FUNCTION "LAnyAxis_UnpubMoveJogPosAxis" : Void   // FC30008, SCL
TITLE = LAnyAxis_UnpubMoveJogPosAxis
{ S7_Optimized_Access := 'TRUE' }
AUTHOR : tech.team.motioncontrol@siemens.com
FAMILY : AnyAxis
VERSION : 1.0
// Support: tech.team.motioncontrol@siemens.com
   VAR_INPUT
      axis : TO_PositioningAxis;   // Axis specification
   END_VAR
   VAR_IN_OUT
      instMC : MC_MOVEJOG;   // Instance of MC_Instruction
   END_VAR
   // Ret_Val : No return value
BEGIN
   // Call of MC_Instruction
   #instMC(Axis := #axis);
END_FUNCTION

FUNCTION "LAnyAxis_UnpubMoveJogSyncAxis" : Void   // FC30010, SCL
TITLE = LAnyAxis_UnpubMoveJogSyncAxis
{ S7_Optimized_Access := 'TRUE' }
AUTHOR : tech.team.motioncontrol@siemens.com
FAMILY : AnyAxis
VERSION : 1.0
// Support: tech.team.motioncontrol@siemens.com
   VAR_INPUT
      axis : TO_SynchronousAxis;   // Axis specification
   END_VAR
   VAR_IN_OUT
      instMC : MC_MOVEJOG;   // Instance of MC_Instruction
   END_VAR
   // Ret_Val : No return value
BEGIN
   // Call of MC_Instruction
   #instMC(Axis := #axis);
END_FUNCTION

// folder: LAnyAxis_Blocks/InternalSubBlocks/MC_MoveRelative

FUNCTION "LAnyAxis_UnpubMoveRelativeSyncAxis" : Void   // FC30012, SCL
TITLE = LAnyAxis_UnpubMoveRelativeSyncAxis
{ S7_Optimized_Access := 'TRUE' }
AUTHOR : tech.team.motioncontrol@siemens.com
FAMILY : AnyAxis
VERSION : 1.0
// Support: tech.team.motioncontrol@siemens.com
   VAR_INPUT
      axis : TO_SynchronousAxis;   // Axis specification
   END_VAR
   VAR_IN_OUT
      instMC : MC_MOVERELATIVE;   // Instance of MC_Instruction
   END_VAR
   // Ret_Val : No return value
BEGIN
   // Call of MC_Instruction
   #instMC(Axis := #axis);
END_FUNCTION

// folder: LAnyAxis_Blocks/InternalSubBlocks/MC_MoveSuperimposed

FUNCTION "LAnyAxis_UnpubMoveSuperimposedSyncAxis" : Void   // FC30014, SCL
TITLE = LAnyAxis_UnpubMoveSuperimposedSyncAxis
{ S7_Optimized_Access := 'TRUE' }
AUTHOR : tech.team.motioncontrol@siemens.com
FAMILY : AnyAxis
VERSION : 1.0
// Support: tech.team.motioncontrol@siemens.com
   VAR_INPUT
      axis : TO_SynchronousAxis;   // Axis specification
   END_VAR
   VAR_IN_OUT
      instMC : MC_MOVESUPERIMPOSED;   // Instance of MC_Instruction
   END_VAR
   // Ret_Val : No return value
BEGIN
   // Call of MC_Instruction
   #instMC(Axis := #axis);
END_FUNCTION

// folder: LAnyAxis_Blocks/InternalSubBlocks/MC_MoveVelocity

FUNCTION "LAnyAxis_UnpubMoveVelocityPosAxis" : Void   // FC30015, SCL
TITLE = LAnyAxis_UnpubMoveVelocityPosAxis
{ S7_Optimized_Access := 'TRUE' }
AUTHOR : tech.team.motioncontrol@siemens.com
FAMILY : AnyAxis
VERSION : 1.0
// Support: tech.team.motioncontrol@siemens.com
   VAR_INPUT
      axis : TO_PositioningAxis;   // Axis specification
   END_VAR
   VAR_IN_OUT
      instMC : MC_MOVEVELOCITY;   // Instance of MC_Instruction
   END_VAR
   // Ret_Val : No return value
BEGIN
   // Call of MC_Instruction
   #instMC(Axis := #axis);
END_FUNCTION

FUNCTION "LAnyAxis_UnpubMoveVelocitySyncAxis" : Void   // FC30017, SCL
TITLE = LAnyAxis_UnpubMoveVelocitySyncAxis
{ S7_Optimized_Access := 'TRUE' }
AUTHOR : tech.team.motioncontrol@siemens.com
FAMILY : AnyAxis
VERSION : 1.0
// Support: tech.team.motioncontrol@siemens.com
   VAR_INPUT
      axis : TO_SynchronousAxis;   // Axis specification
   END_VAR
   VAR_IN_OUT
      instMC : MC_MOVEVELOCITY;   // Instance of MC_Instruction
   END_VAR
   // Ret_Val : No return value
BEGIN
   // Call of MC_Instruction
   #instMC(Axis := #axis);
END_FUNCTION

// folder: LAnyAxis_Blocks/InternalSubBlocks/MC_Power

FUNCTION "LAnyAxis_UnpubPowerExtEncoder" : Void   // FC30018, SCL
TITLE = LAnyAxis_UnpubPowerExtEncoder
{ S7_Optimized_Access := 'TRUE' }
AUTHOR : tech.team.motioncontrol@siemens.com
FAMILY : AnyAxis
VERSION : 1.0
// Support: tech.team.motioncontrol@siemens.com
   VAR_INPUT
      axis : TO_ExternalEncoder;   // Axis specification
   END_VAR
   VAR_IN_OUT
      instMC : MC_POWER;   // Instance of MC_Instruction
   END_VAR
   // Ret_Val : No return value
BEGIN
   // Call of MC_Instruction
   #instMC(Axis := #axis);
END_FUNCTION

FUNCTION "LAnyAxis_UnpubPowerPosAxis" : Void   // FC30019, SCL
TITLE = LAnyAxis_UnpubPowerPosAxis
{ S7_Optimized_Access := 'TRUE' }
AUTHOR : tech.team.motioncontrol@siemens.com
FAMILY : AnyAxis
VERSION : 1.0
// Support: tech.team.motioncontrol@siemens.com
   VAR_INPUT
      axis : TO_PositioningAxis;   // Axis specification
   END_VAR
   VAR_IN_OUT
      instMC : MC_POWER;   // Instance of MC_Instruction
   END_VAR
   // Ret_Val : No return value
BEGIN
   // Call of MC_Instruction
   #instMC(Axis := #axis);
END_FUNCTION

FUNCTION "LAnyAxis_UnpubPowerSpeedAxis" : Void   // FC30020, SCL
TITLE = LAnyAxis_UnpubPowerSpeedAxis
{ S7_Optimized_Access := 'TRUE' }
AUTHOR : tech.team.motioncontrol@siemens.com
FAMILY : AnyAxis
VERSION : 1.0
// Support: tech.team.motioncontrol@siemens.com
   VAR_INPUT
      axis : TO_SpeedAxis;   // Axis specification
   END_VAR
   VAR_IN_OUT
      instMC : MC_POWER;   // Instance of MC_Instruction
   END_VAR
   // Ret_Val : No return value
BEGIN
   // Call of MC_Instruction
   #instMC(Axis := #axis);
END_FUNCTION

FUNCTION "LAnyAxis_UnpubPowerSyncAxis" : Void   // FC30021, SCL
TITLE = LAnyAxis_UnpubPowerSyncAxis
{ S7_Optimized_Access := 'TRUE' }
AUTHOR : tech.team.motioncontrol@siemens.com
FAMILY : AnyAxis
VERSION : 1.0
// Support: tech.team.motioncontrol@siemens.com
   VAR_INPUT
      axis : TO_SynchronousAxis;   // Axis specification
   END_VAR
   VAR_IN_OUT
      instMC : MC_POWER;   // Instance of MC_Instruction
   END_VAR
   // Ret_Val : No return value
BEGIN
   // Call of MC_Instruction
   #instMC(Axis := #axis);
END_FUNCTION

// folder: LAnyAxis_Blocks/InternalSubBlocks/MC_Reset

FUNCTION "LAnyAxis_UnpubResetExtEncoder" : Void   // FC30022, SCL
TITLE = LAnyAxis_UnpubResetExtEncoder
{ S7_Optimized_Access := 'TRUE' }
AUTHOR : tech.team.motioncontrol@siemens.com
FAMILY : AnyAxis
VERSION : 1.0
// Support: tech.team.motioncontrol@siemens.com
   VAR_INPUT
      axis : TO_ExternalEncoder;   // Axis specification
   END_VAR
   VAR_IN_OUT
      instMC : MC_RESET;   // Instance of MC_Instruction
   END_VAR
   // Ret_Val : No return value
BEGIN
   // Call of MC_Instruction
   #instMC(Axis := #axis);
END_FUNCTION

FUNCTION "LAnyAxis_UnpubResetSpeedAxis" : Void   // FC30024, SCL
TITLE = LAnyAxis_UnpubResetSpeedAxis
{ S7_Optimized_Access := 'TRUE' }
AUTHOR : tech.team.motioncontrol@siemens.com
FAMILY : AnyAxis
VERSION : 1.0
// Support: tech.team.motioncontrol@siemens.com
   VAR_INPUT
      axis : TO_SpeedAxis;   // Axis specification
   END_VAR
   VAR_IN_OUT
      instMC : MC_RESET;   // Instance of MC_Instruction
   END_VAR
   // Ret_Val : No return value
BEGIN
   // Call of MC_Instruction
   #instMC(Axis := #axis);
END_FUNCTION

FUNCTION "LAnyAxis_UnpubResetSyncAxis" : Void   // FC30025, SCL
TITLE = LAnyAxis_UnpubResetSyncAxis
{ S7_Optimized_Access := 'TRUE' }
AUTHOR : tech.team.motioncontrol@siemens.com
FAMILY : AnyAxis
VERSION : 1.0
// Support: tech.team.motioncontrol@siemens.com
   VAR_INPUT
      axis : TO_SynchronousAxis;   // Axis specification
   END_VAR
   VAR_IN_OUT
      instMC : MC_RESET;   // Instance of MC_Instruction
   END_VAR
   // Ret_Val : No return value
BEGIN
   // Call of MC_Instruction
   #instMC(Axis := #axis);
END_FUNCTION

FUNCTION "LAnyAxis_UnpubResetProxy" : Void   // FC30057, SCL
TITLE = LAnyAxis_UnpubResetProxy
{ S7_Optimized_Access := 'TRUE' }
AUTHOR : tech.team.motioncontrol@siemens.com
FAMILY : AnyAxis
VERSION : 1.0
// Support: tech.team.motioncontrol@siemens.com
   VAR_INPUT
      axis : TO_LeadingAxisProxy;   // Axis specification
   END_VAR
   VAR_IN_OUT
      instMC : MC_RESET;   // Instance of MC_Instruction
   END_VAR
   // Ret_Val : No return value
BEGIN
   // Call of MC_Instruction
   #instMC(Axis := #axis);
END_FUNCTION

FUNCTION "LAnyAxis_UnpubResetPosAxis" : Void   // FC30071, SCL
TITLE = LAnyAxis_UnpubResetPosAxis
{ S7_Optimized_Access := 'TRUE' }
AUTHOR : tech.team.motioncontrol@siemens.com
FAMILY : AnyAxis
VERSION : 1.0
// Support: tech.team.motioncontrol@siemens.com
   VAR_INPUT
      axis : TO_PositioningAxis;   // Axis specification
   END_VAR
   VAR_IN_OUT
      instMC : MC_RESET;   // Instance of MC_Instruction
   END_VAR
   // Ret_Val : No return value
BEGIN
   // Call of MC_Instruction
   #instMC(Axis := #axis);
END_FUNCTION

// folder: LAnyAxis_Blocks/InternalSubBlocks/MC_SetAxisSTW

FUNCTION "LAnyAxis_UnpubSetAxisSTWPosAxis" : Void   // FC30026, SCL
TITLE = LAnyAxis_UnpubSetAxisSTWPosAxis
{ S7_Optimized_Access := 'TRUE' }
AUTHOR : tech.team.motioncontrol@siemens.com
FAMILY : AnyAxis
VERSION : 1.0
// Support: tech.team.motioncontrol@siemens.com
   VAR_INPUT
      axis : TO_PositioningAxis;   // Axis specification
   END_VAR
   VAR_IN_OUT
      instMC : MC_SETAXISSTW;   // Instance of MC_Instruction
   END_VAR
   // Ret_Val : No return value
BEGIN
   // Call of MC_Instruction
   #instMC(Axis := #axis);
END_FUNCTION

FUNCTION "LAnyAxis_UnpubSetAxisSTWSyncAxis" : Void   // FC30028, SCL
TITLE = LAnyAxis_UnpubSetAxisSTWSyncAxis
{ S7_Optimized_Access := 'TRUE' }
AUTHOR : tech.team.motioncontrol@siemens.com
FAMILY : AnyAxis
VERSION : 1.0
// Support: tech.team.motioncontrol@siemens.com
   VAR_INPUT
      axis : TO_SynchronousAxis;   // Axis specification
   END_VAR
   VAR_IN_OUT
      instMC : MC_SETAXISSTW;   // Instance of MC_Instruction
   END_VAR
   // Ret_Val : No return value
BEGIN
   // Call of MC_Instruction
   #instMC(Axis := #axis);
END_FUNCTION

// folder: LAnyAxis_Blocks/LAnyAxis_MC_SynchronousMotion

FUNCTION_BLOCK "LAnyAxis_MC_GearIn"   // FB30020, SCL
TITLE = LAnyAxis_MC_GearIn
{ S7_Optimized_Access := 'TRUE' }
AUTHOR : tech.team.motioncontrol@siemens.com
FAMILY : AnyAxis
VERSION : 1.0
// Support: tech.team.motioncontrol@siemens.com 
// See corresponding MC_ instruction in TIA Portal help (information system)
   VAR_INPUT
      Master : DB_ANY;   // See corresponding parameter of MC_ instruction in TIA Portal help (information system)
      Slave : DB_ANY;   // See corresponding parameter of MC_ instruction in TIA Portal help (information system)
      Execute : Bool;   // See corresponding parameter of MC_ instruction in TIA Portal help (information system)
      RatioNumerator : DInt := 1;   // See corresponding parameter of MC_ instruction in TIA Portal help (information system)
      RatioDenominator : DInt := 1;   // See corresponding parameter of MC_ instruction in TIA Portal help (information system)
      Acceleration : LReal := -1.0;   // See corresponding parameter of MC_ instruction in TIA Portal help (information system)
      Deceleration : LReal := -1.0;   // See corresponding parameter of MC_ instruction in TIA Portal help (information system)
      Jerk : LReal := -1.0;   // See corresponding parameter of MC_ instruction in TIA Portal help (information system)
   END_VAR
   VAR_OUTPUT
      InGear : Bool;   // See corresponding parameter of MC_ instruction in TIA Portal help (information system)
      Busy : Bool;   // See corresponding parameter of MC_ instruction in TIA Portal help (information system)
      CommandAborted : Bool;   // See corresponding parameter of MC_ instruction in TIA Portal help (information system)
      Error : Bool;   // See corresponding parameter of MC_ instruction in TIA Portal help (information system)
      ErrorID : Word;   // See corresponding parameter of MC_ instruction in TIA Portal help (information system)
   END_VAR
   VAR
      instMC : MC_GEARIN;   // Instance of MC_Instruction
      statExecuteOld : Bool;   // Old value of execute
      statAxis : DB_ANY;   // Internal variable of axis
      statAxisType : Int;   // Actual state / axis type
      statMaster : DB_ANY;   // Internal variable of Master
      statMasterType : Int;   // Type of master axis
   END_VAR
   VAR CONSTANT
      ERROR_INVALID_TECHNOLOGY_OBJECT : Word := 16#8002;   // See corresponding parameter of MC_ instruction in TIA Portal help (information system)
      IDLE : Int := 0;   // State idle
      INVALID_AXIS : Int := -1;   // Axis type: Invalid
      INVALID_MASTER : Int := -2;   // Invalid master type
      EXTERNAL_ENCODER : Int := 1;   // Axis type: External encoder
      POSITIONING_AXIS : Int := 3;   // Axis type: Positioning axis
      SYNCHRONOUS_AXIS : Int := 4;   // Axis type: Synchronous axis
      PROXY : Int := 5;   // Axis type: Leading axis proxy
   END_VAR
BEGIN
   REGION HEADER
     //================================================================================
     // SIEMENS AG
     // (c)Copyright 2020 All Rights Reserved
     //--------------------------------------------------------------------------------
     // Library: LAnyAxis 
     // Tested with: S7-1515T-2 PN
     // Engineering: TIA Portal V16
     // Restrictions: -
     // Requirements: S7-1500T FW 2.8.1
     // Functionality: Conversion DB_ANY --> TO_Axis
     // Support: tech.team.motioncontrol@siemens.com
     // Note: Parameter comments are only available in language 'English (United States)'
     //--------------------------------------------------------------------------------
     // Change log table:
     // Version  Date        Expert in charge  Changes applied
     // 01.00.00 10.03.2020  RS                First released version
     //================================================================================
   END_REGION

   REGION EXECUTE
     IF #Execute AND NOT #statExecuteOld THEN
       // Copy parameter
       #instMC.RatioNumerator := #RatioNumerator;
       #instMC.RatioDenominator := #RatioDenominator;
       #instMC.Acceleration := #Acceleration;
       #instMC.Deceleration := #Deceleration;
       #instMC.Jerk := #Jerk;

       // Check axis type
       CASE TypeOfDB(#Slave) OF
         TO_SYNCHRONOUSAXIS:
           #statAxisType := #SYNCHRONOUS_AXIS;
           #statAxis := #Slave;

           // Check master type
           CASE TypeOfDB(#Master) OF
             TO_POSITIONINGAXIS:
               #statMasterType := #POSITIONING_AXIS;
               #statMaster := #Master;

             TO_SYNCHRONOUSAXIS:
               #statMasterType := #SYNCHRONOUS_AXIS;
               #statMaster := #Master;

             TO_EXTERNALENCODER:
               #statMasterType := #EXTERNAL_ENCODER;
               #statMaster := #Master;

             TO_LEADINGAXISPROXY:
               #statMasterType := #PROXY;
               #statMaster := #Master;
             ELSE
               // Invalid master
               #statMasterType := #INVALID_AXIS;
               #statMaster := 0;

               #statAxisType := #INVALID_MASTER;
           END_CASE;

         ELSE
           #statAxisType := #INVALID_AXIS;
           #statAxis := 0;
       END_CASE;

     ELSIF NOT #Execute AND (#statAxisType < #IDLE) THEN
       #statAxisType := #IDLE;

       // Outputs
       #InGear := FALSE;
       #Busy := FALSE;
       #CommandAborted := FALSE;
       #Error := FALSE;
       #ErrorID := 16#0000;
     END_IF;

     // Edge detection
     #statExecuteOld := #Execute;
   END_REGION

   CASE #statAxisType OF
     #IDLE:
       ;

     #SYNCHRONOUS_AXIS:
       REGION VALID_AXIS
         // Inputs
         #instMC.Execute := #Execute;

         // Call of MC instruction
         CASE #statMasterType OF
           #POSITIONING_AXIS:
             "LAnyAxis_UnpubGearInMasterPosAxis"(slave := #statAxis,
                                                 master := #statMaster,
                                                 instMC := #instMC);
           #SYNCHRONOUS_AXIS:
             "LAnyAxis_UnpubGearInMasterSyncAxis"(slave := #statAxis,
                                                  master := #statMaster,
                                                  instMC := #instMC);
           #EXTERNAL_ENCODER:
             "LAnyAxis_UnpubGearInMasterExtEncoder"(slave := #statAxis,
                                                    master := #statMaster,
                                                    instMC := #instMC);
           #PROXY:
             "LAnyAxis_UnpubGearInMasterProxy"(slave := #statAxis,
                                               master := #statMaster,
                                               instMC := #instMC);
         END_CASE;

         // Outputs
         #InGear := #instMC.InGear;
         #Busy := #instMC.Busy;
         #CommandAborted := #instMC.CommandAborted;
         #Error := #instMC.Error;
         #ErrorID := #instMC.ErrorId;

         // Status of MC instruction
         IF NOT #instMC.Busy
           AND NOT #instMC.CommandAborted
           AND NOT #instMC.Error
         THEN
           // Not active
           #statAxisType := #IDLE;
         END_IF;
       END_REGION

     ELSE
       REGION INVALID_TECHNOLOGY_OBJECT
         // Outputs
         #InGear := FALSE;
         #Busy := FALSE;
         #CommandAborted := FALSE;
         #Error := TRUE;
         #ErrorID := #ERROR_INVALID_TECHNOLOGY_OBJECT;
       END_REGION
   END_CASE;
END_FUNCTION_BLOCK

FUNCTION_BLOCK "LAnyAxis_MC_GearInPos"   // FB30021, SCL
TITLE = LAnyAxis_MC_GearInPos
{ S7_Optimized_Access := 'TRUE' }
AUTHOR : tech.team.motioncontrol@siemens.com
FAMILY : AnyAxis
VERSION : 1.0
// Support: tech.team.motioncontrol@siemens.com 
// See corresponding MC_ instruction in TIA Portal help (information system)
   VAR_INPUT
      Master : DB_ANY;   // See corresponding parameter of MC_ instruction in TIA Portal help (information system)
      Slave : DB_ANY;   // See corresponding parameter of MC_ instruction in TIA Portal help (information system)
      Execute : Bool;   // See corresponding parameter of MC_ instruction in TIA Portal help (information system)
      RatioNumerator : DInt := 1;   // See corresponding parameter of MC_ instruction in TIA Portal help (information system)
      RatioDenominator : DInt := 1;   // See corresponding parameter of MC_ instruction in TIA Portal help (information system)
      MasterSyncPosition : LReal;   // See corresponding parameter of MC_ instruction in TIA Portal help (information system)
      SlaveSyncPosition : LReal;   // See corresponding parameter of MC_ instruction in TIA Portal help (information system)
      SyncProfileReference : DInt := 1;   // See corresponding parameter of MC_ instruction in TIA Portal help (information system)
      MasterStartDistance : LReal := 1.0;   // See corresponding parameter of MC_ instruction in TIA Portal help (information system)
      Velocity : LReal := -1.0;   // See corresponding parameter of MC_ instruction in TIA Portal help (information system)
      Acceleration : LReal := -1.0;   // See corresponding parameter of MC_ instruction in TIA Portal help (information system)
      Deceleration : LReal := -1.0;   // See corresponding parameter of MC_ instruction in TIA Portal help (information system)
      Jerk : LReal := -1.0;   // See corresponding parameter of MC_ instruction in TIA Portal help (information system)
      SyncDirection : DInt := 3;   // See corresponding parameter of MC_ instruction in TIA Portal help (information system)
   END_VAR
   VAR_OUTPUT
      StartSync : Bool;   // See corresponding parameter of MC_ instruction in TIA Portal help (information system)
      InSync : Bool;   // See corresponding parameter of MC_ instruction in TIA Portal help (information system)
      Busy : Bool;   // See corresponding parameter of MC_ instruction in TIA Portal help (information system)
      CommandAborted : Bool;   // See corresponding parameter of MC_ instruction in TIA Portal help (information system)
      Error : Bool;   // See corresponding parameter of MC_ instruction in TIA Portal help (information system)
      ErrorID : Word;   // See corresponding parameter of MC_ instruction in TIA Portal help (information system)
   END_VAR
   VAR
      instMC : MC_GEARINPOS;   // Instance of MC_Instruction
      statExecuteOld : Bool;   // Old value of execute
      statAxis : DB_ANY;   // Internal variable of axis
      statAxisType : Int;   // Actual state / axis type
      statMaster : DB_ANY;   // Internal variable of Master
      statMasterType : Int;   // Type of master axis
   END_VAR
   VAR CONSTANT
      ERROR_INVALID_TECHNOLOGY_OBJECT : Word := 16#8002;   // See corresponding parameter of MC_ instruction in TIA Portal help (information system)
      IDLE : Int := 0;   // State idle
      INVALID_AXIS : Int := -1;   // Axis type: Invalid
      INVALID_MASTER : Int := -2;   // Invalid master type
      EXTERNAL_ENCODER : Int := 1;   // Axis type: External encoder
      POSITIONING_AXIS : Int := 3;   // Axis type: Positioning axis
      SYNCHRONOUS_AXIS : Int := 4;   // Axis type: Synchronous axis
      PROXY : Int := 5;   // Axis type: Leading axis proxy
   END_VAR
BEGIN
   REGION HEADER
     //================================================================================
     // SIEMENS AG
     // (c)Copyright 2020 All Rights Reserved
     //--------------------------------------------------------------------------------
     // Library: LAnyAxis 
     // Tested with: S7-1515T-2 PN
     // Engineering: TIA Portal V16
     // Restrictions: -
     // Requirements: S7-1500T FW 2.8.1
     // Functionality: Conversion DB_ANY --> TO_Axis
     // Support: tech.team.motioncontrol@siemens.com
     // Note: Parameter comments are only available in language 'English (United States)'
     //--------------------------------------------------------------------------------
     // Change log table:
     // Version  Date        Expert in charge  Changes applied
     // 01.00.00 10.03.2020  RS                First released version
     //================================================================================
   END_REGION

   REGION EXECUTE
     IF #Execute AND NOT #statExecuteOld THEN
       // Copy parameter
       #instMC.RatioNumerator := #RatioNumerator;
       #instMC.RatioDenominator := #RatioDenominator;
       #instMC.MasterSyncPosition := #MasterSyncPosition;
       #instMC.SlaveSyncPosition := #SlaveSyncPosition;
       #instMC.SyncProfileReference := #SyncProfileReference;
       #instMC.MasterStartDistance := #MasterStartDistance;
       #instMC.Velocity := #Velocity;
       #instMC.Acceleration := #Acceleration;
       #instMC.Deceleration := #Deceleration;
       #instMC.Jerk := #Jerk;
       #instMC.SyncDirection := #SyncDirection;

       // Check axis type
       CASE TypeOfDB(#Slave) OF
         TO_SYNCHRONOUSAXIS:
           #statAxisType := #SYNCHRONOUS_AXIS;
           #statAxis := #Slave;

           // Check master type
           CASE TypeOfDB(#Master) OF
             TO_POSITIONINGAXIS:
               #statMasterType := #POSITIONING_AXIS;
               #statMaster := #Master;

             TO_SYNCHRONOUSAXIS:
               #statMasterType := #SYNCHRONOUS_AXIS;
               #statMaster := #Master;

             TO_EXTERNALENCODER:
               #statMasterType := #EXTERNAL_ENCODER;
               #statMaster := #Master;

             TO_LEADINGAXISPROXY:
               #statMasterType := #PROXY;
               #statMaster := #Master;
             ELSE
               #statMasterType := #INVALID_AXIS;
               #statMaster := 0;

               // Invalid master
               #statAxisType := #INVALID_MASTER;
           END_CASE;

         ELSE
           #statAxisType := #INVALID_AXIS;
           #statAxis := 0;
       END_CASE;

     ELSIF NOT #Execute AND (#statAxisType < #IDLE) THEN
       #statAxisType := #IDLE;

       // Outputs
       #StartSync := FALSE;
       #InSync := FALSE;
       #Busy := FALSE;
       #CommandAborted := FALSE;
       #Error := FALSE;
       #ErrorID := 16#0000;
     END_IF;

     // Edge detection
     #statExecuteOld := #Execute;
   END_REGION

   CASE #statAxisType OF
     #IDLE:
       ;

     #SYNCHRONOUS_AXIS:
       REGION VALID_AXIS
         // Inputs
         #instMC.Execute := #Execute;

         // Call of MC instruction
         CASE #statMasterType OF
           #POSITIONING_AXIS:
             "LAnyAxis_UnpubGearInPosMasterPosAxis"(slave := #statAxis,
                                                    master := #statMaster,
                                                    instMC := #instMC);
           #SYNCHRONOUS_AXIS:
             "LAnyAxis_UnpubGearInPosMasterSyncAxis"(slave := #statAxis,
                                                     master := #statMaster,
                                                     instMC := #instMC);
           #EXTERNAL_ENCODER:
             "LAnyAxis_UnpubGearInPosMasterExtEncoder"(slave := #statAxis,
                                                       master := #statMaster,
                                                       instMC := #instMC);
           #PROXY:
             "LAnyAxis_UnpubGearInPosMasterProxy"(slave := #statAxis,
                                                  master := #statMaster,
                                                  instMC := #instMC);
         END_CASE;

         // Outputs
         #StartSync := #instMC.StartSync;
         #InSync := #instMC.InSync;
         #Busy := #instMC.Busy;
         #CommandAborted := #instMC.CommandAborted;
         #Error := #instMC.Error;
         #ErrorID := #instMC.ErrorId;

         // Status of MC instruction
         IF NOT #instMC.Busy
           AND NOT #instMC.CommandAborted
           AND NOT #instMC.Error
         THEN
           // Not active
           #statAxisType := #IDLE;
         END_IF;
       END_REGION

     ELSE
       REGION INVALID_TECHNOLOGY_OBJECT
         // Outputs
         #StartSync := FALSE;
         #InSync := FALSE;
         #Busy := FALSE;
         #CommandAborted := FALSE;
         #Error := TRUE;
         #ErrorID := #ERROR_INVALID_TECHNOLOGY_OBJECT;
       END_REGION
   END_CASE;
END_FUNCTION_BLOCK

FUNCTION_BLOCK "LAnyAxis_MC_PhasingRelative"   // FB30022, SCL
TITLE = LAnyAxis_MC_PhasingRelative
{ S7_Optimized_Access := 'TRUE' }
AUTHOR : tech.team.motioncontrol@siemens.com
FAMILY : AnyAxis
VERSION : 1.1
// Support: tech.team.motioncontrol@siemens.com 
// See corresponding MC_ instruction in TIA Portal help (information system)
   VAR_INPUT
      Master : DB_ANY;   // See corresponding parameter of MC_ instruction in TIA Portal help (information system)
      Slave : DB_ANY;   // See corresponding parameter of MC_ instruction in TIA Portal help (information system)
      Execute : Bool;   // See corresponding parameter of MC_ instruction in TIA Portal help (information system)
      PhaseShift : LReal;   // See corresponding parameter of MC_ instruction in TIA Portal help (information system)
      Velocity : LReal := -1.0;   // See corresponding parameter of MC_ instruction in TIA Portal help (information system)
      Acceleration : LReal := -1.0;   // See corresponding parameter of MC_ instruction in TIA Portal help (information system)
      Deceleration : LReal := -1.0;   // See corresponding parameter of MC_ instruction in TIA Portal help (information system)
      Jerk : LReal := -1.0;   // See corresponding parameter of MC_ instruction in TIA Portal help (information system)
      ProfileReference : DInt;   // See corresponding parameter of MC_ instruction in TIA Portal help (information system)
      PhasingDistance : LReal;   // See corresponding parameter of MC_ instruction in TIA Portal help (information system)
      StartPosition : LReal;   // See corresponding parameter of MC_ instruction in TIA Portal help (information system)
      Direction : DInt := 3;   // See corresponding parameter of MC_ instruction in TIA Portal help (information system)
   END_VAR
   VAR_OUTPUT
      Done : Bool;   // See corresponding parameter of MC_ instruction in TIA Portal help (information system)
      Busy : Bool;   // See corresponding parameter of MC_ instruction in TIA Portal help (information system)
      CommandAborted : Bool;   // See corresponding parameter of MC_ instruction in TIA Portal help (information system)
      Error : Bool;   // See corresponding parameter of MC_ instruction in TIA Portal help (information system)
      ErrorID : Word;   // See corresponding parameter of MC_ instruction in TIA Portal help (information system)
      CoveredPhaseShift : LReal;   // See corresponding parameter of MC_ instruction in TIA Portal help (information system)
      StartPhasing : Bool;   // See corresponding parameter of MC_ instruction in TIA Portal help (information system)
   END_VAR
   VAR
      instMC : MC_PHASINGRELATIVE;   // Instance of MC_Instruction
      statExecuteOld : Bool;   // Old value of execute
      statAxis : DB_ANY;   // Internal variable of axis
      statAxisType : Int;   // Actual state / axis type
      statMaster : DB_ANY;   // Internal variable of Master
      statMasterType : Int;   // Type of master axis
   END_VAR
   VAR CONSTANT
      ERROR_INVALID_TECHNOLOGY_OBJECT : Word := 16#8002;   // See corresponding parameter of MC_ instruction in TIA Portal help (information system)
      IDLE : Int := 0;   // State idle
      INVALID_AXIS : Int := -1;   // Axis type: Invalid
      INVALID_MASTER : Int := -2;   // Invalid master type
      EXTERNAL_ENCODER : Int := 1;   // Axis type: External encoder
      POSITIONING_AXIS : Int := 3;   // Axis type: Positioning axis
      SYNCHRONOUS_AXIS : Int := 4;   // Axis type: Synchronous axis
      PROXY : Int := 5;   // Axis type: Leading axis proxy
   END_VAR
BEGIN
   REGION HEADER
     //================================================================================
     // SIEMENS AG
     // (c)Copyright 2021 All Rights Reserved
     //--------------------------------------------------------------------------------
     // Library: LAnyAxis 
     // Tested with: S7-1515T-2 PN
     // Engineering: TIA Portal V17
     // Restrictions: -
     // Requirements: S7-1500T FW 2.9
     // Functionality: Conversion DB_ANY --> TO_Axis
     // Support: tech.team.motioncontrol@siemens.com
     // Note: Parameter comments are only available in language 'English (United States)'
     //--------------------------------------------------------------------------------
     // Change log table:
     // Version  Date        Expert in charge  Changes applied
     // 01.00.00 10.03.2020  RS                First released version
     // 01.01.00 24.02.2021  RS                Update MC V6.0
     //================================================================================
   END_REGION

   REGION EXECUTE
     IF #Execute AND NOT #statExecuteOld THEN
       // Copy parameter
       #instMC.PhaseShift       := #PhaseShift;
       #instMC.Velocity         := #Velocity;
       #instMC.Acceleration     := #Acceleration;
       #instMC.Deceleration     := #Deceleration;
       #instMC.Jerk             := #Jerk;
       #instMC.ProfileReference := #ProfileReference;
       #instMC.PhasingDistance  := #PhasingDistance;
       #instMC.StartPosition    := #StartPosition;
       #instMC.Direction        := #Direction;

       // Check axis type
       CASE TypeOfDB(#Slave) OF
         TO_SYNCHRONOUSAXIS:
           #statAxisType := #SYNCHRONOUS_AXIS;
           #statAxis := #Slave;

           // Check master type
           CASE TypeOfDB(#Master) OF
             TO_POSITIONINGAXIS:
               #statMasterType := #POSITIONING_AXIS;
               #statMaster := #Master;

             TO_SYNCHRONOUSAXIS:
               #statMasterType := #SYNCHRONOUS_AXIS;
               #statMaster := #Master;

             TO_EXTERNALENCODER:
               #statMasterType := #EXTERNAL_ENCODER;
               #statMaster := #Master;

             TO_LEADINGAXISPROXY:
               #statMasterType := #PROXY;
               #statMaster := #Master;
             ELSE
               #statMasterType := #INVALID_AXIS;
               #statMaster := 0;

               // Invalid master
               #statAxisType := #INVALID_MASTER;
           END_CASE;

         ELSE
           #statAxisType := #INVALID_AXIS;
           #statAxis := 0;
       END_CASE;

     ELSIF NOT #Execute AND (#statAxisType < #IDLE) THEN
       #statAxisType := #IDLE;

       // Outputs
       #Done              := FALSE;
       #Busy              := FALSE;
       #CommandAborted    := FALSE;
       #Error             := FALSE;
       #ErrorID           := 16#0000;
       #CoveredPhaseShift := 0.0;
       #StartPhasing      := FALSE;
     END_IF;

     // Edge detection
     #statExecuteOld := #Execute;
   END_REGION

   CASE #statAxisType OF
     #IDLE:
       ;

     #SYNCHRONOUS_AXIS:
       REGION VALID_AXIS
         // Inputs  
         #instMC.Execute := #Execute;

         // Call of MC instruction
         CASE #statMasterType OF
           #POSITIONING_AXIS:
             "LAnyAxis_UnpubPhasingRelativeMasterPosAxis"(slave  := #statAxis,
                                                          master := #statMaster,
                                                          instMC := #instMC);
           #SYNCHRONOUS_AXIS:
             "LAnyAxis_UnpubPhasingRelativeMasterSyncAxis"(slave  := #statAxis,
                                                           master := #statMaster,
                                                           instMC := #instMC);
           #EXTERNAL_ENCODER:
             "LAnyAxis_UnpubPhasingRelativeMasterExtEncoder"(slave  := #statAxis,
                                                             master := #statMaster,
                                                             instMC := #instMC);
           #PROXY:
             "LAnyAxis_UnpubPhasingRelativeMasterProxy"(slave  := #statAxis,
                                                        master := #statMaster,
                                                        instMC := #instMC);
         END_CASE;

         // Outputs
         #Done              := #instMC.Done;
         #Busy              := #instMC.Busy;
         #CommandAborted    := #instMC.CommandAborted;
         #Error             := #instMC.Error;
         #ErrorID           := #instMC.ErrorId;
         #CoveredPhaseShift := #instMC.CoveredPhaseShift;
         #StartPhasing      := #instMC.StartPhasing;

         // Status of MC instruction
         IF NOT #instMC.Done
           AND NOT #instMC.Busy
           AND NOT #instMC.CommandAborted
           AND NOT #instMC.Error
         THEN
           // Not active
           #statAxisType := #IDLE;
         END_IF;
       END_REGION

     ELSE
       REGION INVALID_TECHNOLOGY_OBJECT
         // Outputs
         #Done              := FALSE;
         #Busy              := FALSE;
         #CommandAborted    := FALSE;
         #Error             := TRUE;
         #ErrorID           := #ERROR_INVALID_TECHNOLOGY_OBJECT;
         #CoveredPhaseShift := 0.0;
         #StartPhasing      := FALSE;
       END_REGION
   END_CASE;
END_FUNCTION_BLOCK

FUNCTION_BLOCK "LAnyAxis_MC_PhasingAbsolute"   // FB30023, SCL
TITLE = LAnyAxis_MC_PhasingAbsolute
{ S7_Optimized_Access := 'TRUE' }
AUTHOR : tech.team.motioncontrol@siemens.com
FAMILY : AnyAxis
VERSION : 1.1
// Support: tech.team.motioncontrol@siemens.com 
// See corresponding MC_ instruction in TIA Portal help (information system)
   VAR_INPUT
      Master : DB_ANY;   // See corresponding parameter of MC_ instruction in TIA Portal help (information system)
      Slave : DB_ANY;   // See corresponding parameter of MC_ instruction in TIA Portal help (information system)
      Execute : Bool;   // See corresponding parameter of MC_ instruction in TIA Portal help (information system)
      PhaseShift : LReal;   // See corresponding parameter of MC_ instruction in TIA Portal help (information system)
      Velocity : LReal := -1.0;   // See corresponding parameter of MC_ instruction in TIA Portal help (information system)
      Acceleration : LReal := -1.0;   // See corresponding parameter of MC_ instruction in TIA Portal help (information system)
      Deceleration : LReal := -1.0;   // See corresponding parameter of MC_ instruction in TIA Portal help (information system)
      Jerk : LReal := -1.0;   // See corresponding parameter of MC_ instruction in TIA Portal help (information system)
      ProfileReference : DInt;   // See corresponding parameter of MC_ instruction in TIA Portal help (information system)
      PhasingDistance : LReal;   // See corresponding parameter of MC_ instruction in TIA Portal help (information system)
      StartPosition : LReal;   // See corresponding parameter of MC_ instruction in TIA Portal help (information system)
      Direction : DInt := 3;   // See corresponding parameter of MC_ instruction in TIA Portal help (information system)
   END_VAR
   VAR_OUTPUT
      Done : Bool;   // See corresponding parameter of MC_ instruction in TIA Portal help (information system)
      Busy : Bool;   // See corresponding parameter of MC_ instruction in TIA Portal help (information system)
      CommandAborted : Bool;   // See corresponding parameter of MC_ instruction in TIA Portal help (information system)
      Error : Bool;   // See corresponding parameter of MC_ instruction in TIA Portal help (information system)
      ErrorID : Word;   // See corresponding parameter of MC_ instruction in TIA Portal help (information system)
      AbsolutePhaseShift : LReal;   // See corresponding parameter of MC_ instruction in TIA Portal help (information system)
      StartPhasing : Bool;   // See corresponding parameter of MC_ instruction in TIA Portal help (information system)
   END_VAR
   VAR
      instMC : MC_PHASINGABSOLUTE;   // Instance of MC_Instruction
      statExecuteOld : Bool;   // Old value of execute
      statAxis : DB_ANY;   // Internal variable of axis
      statAxisType : Int;   // Actual state / axis type
      statMaster : DB_ANY;   // Internal variable of Master
      statMasterType : Int;   // Type of master axis
   END_VAR
   VAR CONSTANT
      ERROR_INVALID_TECHNOLOGY_OBJECT : Word := 16#8002;   // See corresponding parameter of MC_ instruction in TIA Portal help (information system)
      IDLE : Int := 0;   // State idle
      INVALID_AXIS : Int := -1;   // Axis type: Invalid
      INVALID_MASTER : Int := -2;   // Invalid master type
      EXTERNAL_ENCODER : Int := 1;   // Axis type: External encoder
      POSITIONING_AXIS : Int := 3;   // Axis type: Positioning axis
      SYNCHRONOUS_AXIS : Int := 4;   // Axis type: Synchronous axis
      PROXY : Int := 5;   // Axis type: Leading axis proxy
   END_VAR
BEGIN
   REGION HEADER
     //================================================================================
     // SIEMENS AG
     // (c)Copyright 2021 All Rights Reserved
     //--------------------------------------------------------------------------------
     // Library: LAnyAxis 
     // Tested with: S7-1515T-2 PN
     // Engineering: TIA Portal V17
     // Restrictions: -
     // Requirements: S7-1500T FW 2.9 
     // Functionality: Conversion DB_ANY --> TO_Axis
     // Support: tech.team.motioncontrol@siemens.com
     // Note: Parameter comments are only available in language 'English (United States)'
     //--------------------------------------------------------------------------------
     // Change log table:
     // Version  Date        Expert in charge  Changes applied
     // 01.00.00 10.03.2020  RS                First released version
     // 01.01.00 24.02.2021  RS                Update MC V6.0
     //================================================================================
   END_REGION

   REGION EXECUTE
     IF #Execute AND NOT #statExecuteOld THEN
       // Copy parameter
       #instMC.PhaseShift       := #PhaseShift;
       #instMC.Velocity         := #Velocity;
       #instMC.Acceleration     := #Acceleration;
       #instMC.Deceleration     := #Deceleration;
       #instMC.Jerk             := #Jerk;
       #instMC.ProfileReference := #ProfileReference;
       #instMC.PhasingDistance  := #PhasingDistance;
       #instMC.StartPosition    := #StartPosition;
       #instMC.Direction        := #Direction;

       // Check axis type
       CASE TypeOfDB(#Slave) OF
         TO_SYNCHRONOUSAXIS:
           #statAxisType := #SYNCHRONOUS_AXIS;
           #statAxis := #Slave;

           // Check master type
           CASE TypeOfDB(#Master) OF
             TO_POSITIONINGAXIS:
               #statMasterType := #POSITIONING_AXIS;
               #statMaster := #Master;

             TO_SYNCHRONOUSAXIS:
               #statMasterType := #SYNCHRONOUS_AXIS;
               #statMaster := #Master;

             TO_EXTERNALENCODER:
               #statMasterType := #EXTERNAL_ENCODER;
               #statMaster := #Master;

             TO_LEADINGAXISPROXY:
               #statMasterType := #PROXY;
               #statMaster := #Master;
             ELSE
               #statMasterType := #INVALID_AXIS;
               #statMaster := 0;

               // Invalid master
               #statAxisType := #INVALID_MASTER;
           END_CASE;

         ELSE
           #statAxisType := #INVALID_AXIS;
           #statAxis := 0;
       END_CASE;

     ELSIF NOT #Execute AND (#statAxisType < #IDLE) THEN
       #statAxisType := #IDLE;

       // Outputs
       #Done               := FALSE;
       #Busy               := FALSE;
       #CommandAborted     := FALSE;
       #Error              := FALSE;
       #ErrorID            := 16#0000;
       #AbsolutePhaseShift := 0.0;
       #StartPhasing       := FALSE;
     END_IF;

     // Edge detection
     #statExecuteOld := #Execute;
   END_REGION

   CASE #statAxisType OF
     #IDLE:
       ;

     #SYNCHRONOUS_AXIS:
       REGION VALID_AXIS
         // Inputs 
         #instMC.Execute := #Execute;

         // Call of MC instruction
         CASE #statMasterType OF
           #POSITIONING_AXIS:
             "LAnyAxis_UnpubPhasingAbsoluteMasterPosAxis"(slave := #statAxis,
                                                          master := #statMaster,
                                                          instMC := #instMC);
           #SYNCHRONOUS_AXIS:
             "LAnyAxis_UnpubPhasingAbsoluteMasterSyncAxis"(slave := #statAxis,
                                                           master := #statMaster,
                                                           instMC := #instMC);
           #EXTERNAL_ENCODER:
             "LAnyAxis_UnpubPhasingAbsoluteMasterExtEncoder"(slave := #statAxis,
                                                             master := #statMaster,
                                                             instMC := #instMC);
           #PROXY:
             "LAnyAxis_UnpubPhasingAbsoluteMasterProxy"(slave := #statAxis,
                                                        master := #statMaster,
                                                        instMC := #instMC);
         END_CASE;

         // Outputs
         #Done               := #instMC.Done;
         #Busy               := #instMC.Busy;
         #CommandAborted     := #instMC.CommandAborted;
         #Error              := #instMC.Error;
         #ErrorID            := #instMC.ErrorId;
         #AbsolutePhaseShift := #instMC.AbsolutePhaseShift;
         #StartPhasing       := #instMC.StartPhasing;

         // Status of MC instruction
         IF NOT #instMC.Done
           AND NOT #instMC.Busy
           AND NOT #instMC.CommandAborted
           AND NOT #instMC.Error
         THEN
           // Not active
           #statAxisType := #IDLE;
         END_IF;
       END_REGION

     ELSE
       REGION INVALID_TECHNOLOGY_OBJECT
         // Outputs
         #Done               := FALSE;
         #Busy               := FALSE;
         #CommandAborted     := FALSE;
         #Error              := TRUE;
         #ErrorID            := #ERROR_INVALID_TECHNOLOGY_OBJECT;
         #AbsolutePhaseShift := 0.0;
         #StartPhasing       := FALSE;
       END_REGION
   END_CASE;
END_FUNCTION_BLOCK

FUNCTION_BLOCK "LAnyAxis_MC_CamIn"   // FB30024, SCL
TITLE = LAnyAxis_MC_CamIn
{ S7_Optimized_Access := 'TRUE' }
AUTHOR : tech.team.motioncontrol@siemens.com
FAMILY : AnyAxis
VERSION : 1.1
// Support: tech.team.motioncontrol@siemens.com 
// See corresponding MC_ instruction in TIA Portal help (information system)
   VAR_INPUT
      Master : DB_ANY;   // See corresponding parameter of MC_ instruction in TIA Portal help (information system)
      Slave : DB_ANY;   // See corresponding parameter of MC_ instruction in TIA Portal help (information system)
      Cam : DB_ANY;   // See corresponding parameter of MC_ instruction in TIA Portal help (information system)
      Execute : Bool;   // See corresponding parameter of MC_ instruction in TIA Portal help (information system)
      MasterOffset : LReal;   // See corresponding parameter of MC_ instruction in TIA Portal help (information system)
      SlaveOffset : LReal;   // See corresponding parameter of MC_ instruction in TIA Portal help (information system)
      MasterScaling : LReal := 1.0;   // See corresponding parameter of MC_ instruction in TIA Portal help (information system)
      SlaveScaling : LReal := 1.0;   // See corresponding parameter of MC_ instruction in TIA Portal help (information system)
      MasterSyncPosition : LReal;   // See corresponding parameter of MC_ instruction in TIA Portal help (information system)
      SyncProfileReference : DInt := 1;   // See corresponding parameter of MC_ instruction in TIA Portal help (information system)
      MasterStartDistance : LReal;   // See corresponding parameter of MC_ instruction in TIA Portal help (information system)
      Velocity : LReal := -1.0;   // See corresponding parameter of MC_ instruction in TIA Portal help (information system)
      Acceleration : LReal := -1.0;   // See corresponding parameter of MC_ instruction in TIA Portal help (information system)
      Deceleration : LReal := -1.0;   // See corresponding parameter of MC_ instruction in TIA Portal help (information system)
      Jerk : LReal := -1.0;   // See corresponding parameter of MC_ instruction in TIA Portal help (information system)
      ApplicationMode : DInt;   // See corresponding parameter of MC_ instruction in TIA Portal help (information system)
      SyncDirection : DInt := 3;   // See corresponding parameter of MC_ instruction in TIA Portal help (information system)
   END_VAR
   VAR_OUTPUT
      StartSync : Bool;   // See corresponding parameter of MC_ instruction in TIA Portal help (information system)
      InSync : Bool;   // See corresponding parameter of MC_ instruction in TIA Portal help (information system)
      Busy : Bool;   // See corresponding parameter of MC_ instruction in TIA Portal help (information system)
      CommandAborted : Bool;   // See corresponding parameter of MC_ instruction in TIA Portal help (information system)
      Error : Bool;   // See corresponding parameter of MC_ instruction in TIA Portal help (information system)
      ErrorID : Word;   // See corresponding parameter of MC_ instruction in TIA Portal help (information system)
      EndOfProfile : Bool;   // See corresponding parameter of MC_ instruction in TIA Portal help (information system)
   END_VAR
   VAR
      instMC : MC_CAMIN;   // Instance of MC_Instruction
      statExecuteOld : Bool;   // Old value of execute
      statAxis : DB_ANY;   // Internal variable of axis
      statAxisType : Int;   // Actual state / axis type
      statMaster : DB_ANY;   // Internal variable of master
      statMasterType : Int;   // Type of master axis
      statCam : DB_ANY;   // Internal variable of cam
      statCamType : Int;   // Type of cam
   END_VAR
   VAR CONSTANT
      ERROR_INVALID_TECHNOLOGY_OBJECT : Word := 16#8002;   // See corresponding parameter of MC_ instruction in TIA Portal help (information system)
      IDLE : Int := 0;   // State idle
      INVALID_AXIS : Int := -1;   // Axis type: Invalid
      INVALID_MASTER : Int := -2;   // Invalid master type
      INVALID_CAM : Int := -3;   // Invalid cam
      EXTERNAL_ENCODER : Int := 1;   // Axis type: External encoder
      POSITIONING_AXIS : Int := 3;   // Axis type: Positioning axis
      SYNCHRONOUS_AXIS : Int := 4;   // Axis type: Synchronous axis
      CAM_1K : Int;   // Cam type: Cam
      CAM_10K : Int := 1;   // Cam type: Cam_10k
      PROXY : Int := 5;   // Axis type: Leading axis proxy
   END_VAR
BEGIN
   REGION HEADER
     //================================================================================
     // SIEMENS AG
     // (c)Copyright 2021 All Rights Reserved
     //--------------------------------------------------------------------------------
     // Library: LAnyAxis 
     // Tested with: S7-1515T-2 PN
     // Engineering: TIA Portal V17
     // Restrictions: -
     // Requirements: S7-1500T FW 2.9
     // Functionality: Conversion DB_ANY --> TO_Axis
     // Support: tech.team.motioncontrol@siemens.com
     // Note: Parameter comments are only available in language 'English (United States)'
     //--------------------------------------------------------------------------------
     // Change log table:
     // Version  Date        Expert in charge  Changes applied
     // 01.00.00 10.03.2020  RS                First released version
     // 01.01.00 24.02.2021  RS                Update MC V6.0
     //================================================================================
   END_REGION

   REGION EXECUTE
     IF #Execute AND NOT #statExecuteOld THEN
       // Copy parameter
       #instMC.MasterOffset         := #MasterOffset;
       #instMC.SlaveOffset          := #SlaveOffset;
       #instMC.MasterScaling        := #MasterScaling;
       #instMC.SlaveScaling         := #SlaveScaling;
       #instMC.MasterSyncPosition   := #MasterSyncPosition;
       #instMC.SyncProfileReference := #SyncProfileReference;
       #instMC.MasterStartDistance  := #MasterStartDistance;
       #instMC.Velocity             := #Velocity;
       #instMC.Acceleration         := #Acceleration;
       #instMC.Deceleration         := #Deceleration;
       #instMC.Jerk                 := #Jerk;
       #instMC.ApplicationMode      := #ApplicationMode;
       #instMC.SyncDirection        := #SyncDirection;

       // Check axis type
       CASE TypeOfDB(#Slave) OF
         TO_SYNCHRONOUSAXIS:
           #statAxisType := #SYNCHRONOUS_AXIS;
           #statAxis := #Slave;

           // Check master type
           CASE TypeOfDB(#Master) OF
             TO_POSITIONINGAXIS:
               #statMasterType := #POSITIONING_AXIS;
               #statMaster := #Master;

             TO_SYNCHRONOUSAXIS:
               #statMasterType := #SYNCHRONOUS_AXIS;
               #statMaster := #Master;

             TO_EXTERNALENCODER:
               #statMasterType := #EXTERNAL_ENCODER;
               #statMaster := #Master;

             TO_LEADINGAXISPROXY:
               #statMasterType := #PROXY;
               #statMaster := #Master;
             ELSE
               #statMasterType := #INVALID_AXIS;
               #statMaster := 0;

               // Invalid master
               #statAxisType := #INVALID_MASTER;
           END_CASE;

         ELSE
           #statAxisType := #INVALID_AXIS;
           #statAxis := 0;
       END_CASE;

       CASE TypeOfDB(#Cam) OF
         TO_CAM:
           #statCam := #Cam;
           #statCamType := #CAM_1K;

         TO_CAM_10K:
           #statCam := #Cam;
           #statCamType := #CAM_10K;

         ELSE
           #statCam := 0;
           #statAxisType := #INVALID_CAM;
       END_CASE;

     ELSIF NOT #Execute AND (#statAxisType < #IDLE) THEN
       #statAxisType := #IDLE;

       // Outputs
       #StartSync      := FALSE;
       #InSync         := FALSE;
       #Busy           := FALSE;
       #CommandAborted := FALSE;
       #Error          := FALSE;
       #ErrorID        := 16#0000;
       #EndOfProfile   := FALSE;
     END_IF;

     // Edge detection
     #statExecuteOld := #Execute;
   END_REGION

   CASE #statAxisType OF
     #IDLE:
       ;

     #SYNCHRONOUS_AXIS:
       REGION VALID_AXIS
         // Inputs 
         #instMC.Execute := #Execute;

         // Call of MC instruction
         CASE #statMasterType OF
           #POSITIONING_AXIS:
             CASE #statCamType OF
               #CAM_1K:
                 "LAnyAxis_UnpubCamInMasterPosAxis"(slave  := #statAxis,
                                                    master := #statMaster,
                                                    cam    := #statCam,
                                                    instMC := #instMC);
               #CAM_10K:
                 "LAnyAxis_UnpubCamIn10kMasterPosAxis"(slave  := #statAxis,
                                                       master := #statMaster,
                                                       cam    := #statCam,
                                                       instMC := #instMC);
             END_CASE;

           #SYNCHRONOUS_AXIS:
             CASE #statCamType OF
               #CAM_1K:
                 "LAnyAxis_UnpubCamInMasterSyncAxis"(slave  := #statAxis,
                                                     master := #statMaster,
                                                     cam    := #statCam,
                                                     instMC := #instMC);

               #CAM_10K:
                 "LAnyAxis_UnpubCamIn10kMasterSyncAxis"(slave  := #statAxis,
                                                        master := #statMaster,
                                                        cam    := #statCam,
                                                        instMC := #instMC);
             END_CASE;

           #EXTERNAL_ENCODER:
             CASE #statCamType OF
               #CAM_1K:
                 "LAnyAxis_UnpubCamInMasterExtEncoder"(slave  := #statAxis,
                                                       master := #statMaster,
                                                       cam    := #statCam,
                                                       instMC := #instMC);

               #CAM_10K:
                 "LAnyAxis_UnpubCamIn10kMasterExtEncoder"(slave  := #statAxis,
                                                          master := #statMaster,
                                                          cam    := #statCam,
                                                          instMC := #instMC);
             END_CASE;

           #PROXY:
             CASE #statCamType OF
               #CAM_1K:
                 "LAnyAxis_UnpubCamInMasterProxy"(slave  := #statAxis,
                                                  master := #statMaster,
                                                  cam    := #statCam,
                                                  instMC := #instMC);

               #CAM_10K:
                 "LAnyAxis_UnpubCamIn10kMasterProxy"(slave  := #statAxis,
                                                     master := #statMaster,
                                                     cam    := #statCam,
                                                     instMC := #instMC);
             END_CASE;
         END_CASE;

         // Outputs
         #StartSync      := #instMC.StartSync;
         #InSync         := #instMC.InSync;
         #Busy           := #instMC.Busy;
         #CommandAborted := #instMC.CommandAborted;
         #Error          := #instMC.Error;
         #ErrorID        := #instMC.ErrorId;
         #EndOfProfile   := #instMC.EndOfProfile;

         // Status of MC instruction
         IF NOT #instMC.Busy
           AND NOT #instMC.CommandAborted
           AND NOT #instMC.Error
           AND NOT #instMC.EndOfProfile
         THEN
           // Not active
           #statAxisType := #IDLE;
         END_IF;
       END_REGION
     ELSE
       REGION INVALID_TECHNOLOGY_OBJECT
         // Outputs
         #StartSync      := FALSE;
         #InSync         := FALSE;
         #Busy           := FALSE;
         #CommandAborted := FALSE;
         #Error          := TRUE;
         #ErrorID        := #ERROR_INVALID_TECHNOLOGY_OBJECT;
         #EndOfProfile   := FALSE;
       END_REGION
   END_CASE;
END_FUNCTION_BLOCK

FUNCTION_BLOCK "LAnyAxis_MC_SynchronizedMotionSimulation"   // FB30025, SCL
TITLE = LAnyAxis_MC_SynchronizedMotionSimulation
{ S7_Optimized_Access := 'TRUE' }
AUTHOR : tech.team.motioncontrol@siemens.com
FAMILY : AnyAxis
VERSION : 1.0
// Support: tech.team.motioncontrol@siemens.com 
// See corresponding MC_ instruction in TIA Portal help (information system)
   VAR_INPUT
      Slave : DB_ANY;   // See corresponding parameter of MC_ instruction in TIA Portal help (information system)
      Enable : Bool;   // See corresponding parameter of MC_ instruction in TIA Portal help (information system)
   END_VAR
   VAR_OUTPUT
      InSimulation : Bool;   // See corresponding parameter of MC_ instruction in TIA Portal help (information system)
      Busy : Bool;   // See corresponding parameter of MC_ instruction in TIA Portal help (information system)
      Error : Bool;   // See corresponding parameter of MC_ instruction in TIA Portal help (information system)
      ErrorID : Word;   // See corresponding parameter of MC_ instruction in TIA Portal help (information system)
   END_VAR
   VAR
      instMC : MC_SYNCHRONIZEDMOTIONSIMULATION;   // Instance of MC_Instruction
      statAxis : DB_ANY;   // Internal variable of axis
      statAxisType : Int;   // Actual state / axis type
   END_VAR
   VAR CONSTANT
      ERROR_INVALID_TECHNOLOGY_OBJECT : Word := 16#8002;   // See corresponding parameter of MC_ instruction in TIA Portal help (information system)
      IDLE : Int := 0;   // State idle
      INVALID_AXIS : Int := -1;   // Axis type: Invalid
      SYNCHRONOUS_AXIS : Int := 4;   // Axis type: Synchronous axis
   END_VAR
BEGIN
   REGION HEADER
     //================================================================================
     // SIEMENS AG
     // (c)Copyright 2020 All Rights Reserved
     //--------------------------------------------------------------------------------
     // Library: LAnyAxis 
     // Tested with: S7-1515T-2 PN
     // Engineering: TIA Portal V16
     // Restrictions: -
     // Requirements: S7-1500T FW 2.8.1
     // Functionality: Conversion DB_ANY --> TO_Axis
     // Support: tech.team.motioncontrol@siemens.com
     // Note: Parameter comments are only available in language 'English (United States)'
     //--------------------------------------------------------------------------------
     // Change log table:
     // Version  Date        Expert in charge  Changes applied
     // 01.00.00 10.03.2020  RS                First released version
     //================================================================================
   END_REGION

   REGION ENABLE
     IF (#statAxisType = #IDLE) AND #Enable THEN
       // check axis type
       CASE TypeOfDB(#Slave) OF
         TO_SYNCHRONOUSAXIS:
           #statAxisType := #SYNCHRONOUS_AXIS;
           #statAxis := #Slave;
         ELSE
           #statAxisType := #INVALID_AXIS;
           #statAxis := 0;
       END_CASE;

     ELSIF NOT #Enable AND (#statAxisType = #INVALID_AXIS) THEN
       #statAxisType := #IDLE;

       // Outputs
       #InSimulation := FALSE;
       #Busy := FALSE;
       #Error := FALSE;
       #ErrorID := 16#0000;
     END_IF;
   END_REGION

   CASE #statAxisType OF
     #IDLE:
       ;

     #SYNCHRONOUS_AXIS:
       REGION SYNCHRONOUS_AXIS
         // Inputs
         #instMC.Enable := #Enable;

         // Call of MC instruction
         #instMC(Slave := #statAxis);

         // Outputs
         #InSimulation := #instMC.InSimulation;
         #Busy := #instMC.Busy;
         #Error := #instMC.Error;
         #ErrorID := #instMC.ErrorId;

         // Status of MC instruction
         IF NOT #instMC.Busy
           AND NOT #instMC.Error
         THEN
           // Not active
           #statAxisType := #IDLE;
         END_IF;
       END_REGION

     ELSE
       REGION INVALID_AXIS
         // Outputs
         #InSimulation := FALSE;
         #Busy := FALSE;
         #Error := TRUE;
         #ErrorID := #ERROR_INVALID_TECHNOLOGY_OBJECT;
       END_REGION
   END_CASE;
END_FUNCTION_BLOCK

FUNCTION_BLOCK "LAnyAxis_MC_OffsetRelative"   // FB30028, SCL
TITLE = LAnyAxis_MC_OffsetRelative
{ S7_Optimized_Access := 'TRUE' }
AUTHOR : tech.team.motioncontrol@siemens.com
FAMILY : AnyAxis
VERSION : 1.1
// Support: tech.team.motioncontrol@siemens.com 
// See corresponding MC_ instruction in TIA Portal help (information system)
   VAR_INPUT
      Slave : DB_ANY;   // See corresponding parameter of MC_ instruction in TIA Portal help (information system)
      Execute : Bool;   // See corresponding parameter of MC_ instruction in TIA Portal help (information system)
      Offset : LReal;   // See corresponding parameter of MC_ instruction in TIA Portal help (information system)
      ProfileReference : DInt := 1;   // See corresponding parameter of MC_ instruction in TIA Portal help (information system)
      OffsetDistance : LReal;   // See corresponding parameter of MC_ instruction in TIA Portal help (information system)
      StartPosition : LReal;   // See corresponding parameter of MC_ instruction in TIA Portal help (information system)
      Direction : DInt := 3;   // See corresponding parameter of MC_ instruction in TIA Portal help (information system)
   END_VAR
   VAR_OUTPUT
      Done : Bool;   // See corresponding parameter of MC_ instruction in TIA Portal help (information system)
      Busy : Bool;   // See corresponding parameter of MC_ instruction in TIA Portal help (information system)
      CommandAborted : Bool;   // See corresponding parameter of MC_ instruction in TIA Portal help (information system)
      Error : Bool;   // See corresponding parameter of MC_ instruction in TIA Portal help (information system)
      ErrorID : Word;   // See corresponding parameter of MC_ instruction in TIA Portal help (information system)
      CoveredOffset : LReal;   // See corresponding parameter of MC_ instruction in TIA Portal help (information system)
      StartOffset : Bool;   // See corresponding parameter of MC_ instruction in TIA Portal help (information system)
   END_VAR
   VAR
      instMC : MC_OFFSETRELATIVE;   // Instance of MC_Instruction
      statExecuteOld : Bool;   // Old value of execute
      statAxis : DB_ANY;   // Internal variable of axis
      statAxisType : Int;   // Actual state / axis type
   END_VAR
   VAR CONSTANT
      ERROR_INVALID_TECHNOLOGY_OBJECT : Word := 16#8002;   // See corresponding parameter of MC_ instruction in TIA Portal help (information system)
      IDLE : Int := 0;   // State idle
      INVALID_AXIS : Int := -1;   // Axis type: Invalid
      SYNCHRONOUS_AXIS : Int := 4;   // Axis type: Synchronous axis
   END_VAR
BEGIN
   REGION HEADER
     //================================================================================
     // SIEMENS AG
     // (c)Copyright 2021 All Rights Reserved
     //--------------------------------------------------------------------------------
     // Library: LAnyAxis 
     // Tested with: S7-1515T-2 PN
     // Engineering: TIA Portal V17
     // Restrictions: -
     // Requirements: S7-1500T FW 2.9
     // Functionality: Conversion DB_ANY --> TO_Axis
     // Support: tech.team.motioncontrol@siemens.com
     // Note: Parameter comments are only available in language 'English (United States)'
     //--------------------------------------------------------------------------------
     // Change log table:
     // Version  Date        Expert in charge  Changes applied
     // 01.00.00 01.01.2021  RS                First released version
     // 01.01.00 24.02.2021  RS                Update MC V6.0
     //================================================================================
   END_REGION

   REGION EXECUTE
     IF #Execute AND NOT #statExecuteOld THEN
       // Copy parameter
         #instMC.Offset           := #Offset;
         #instMC.ProfileReference := #ProfileReference;
         #instMC.OffsetDistance   := #OffsetDistance;
         #instMC.StartPosition    := #StartPosition;
         #instMC.Direction        := #Direction;

       // Check axis type
       CASE TypeOfDB(#Slave) OF
         TO_SYNCHRONOUSAXIS:
           #statAxisType := #SYNCHRONOUS_AXIS;
           #statAxis := #Slave;
       ELSE
           #statAxisType := #INVALID_AXIS;
           #statAxis := 0;
       END_CASE;

     ELSIF NOT #Execute AND (#statAxisType < #IDLE) THEN
       #statAxisType := #IDLE;

       // Outputs
       #Done           := FALSE;
       #Busy           := FALSE;
       #CommandAborted := FALSE;
       #Error          := FALSE;
       #ErrorID        := 16#0000;
       #CoveredOffset  := 0.0;
       #StartOffset    := FALSE;
     END_IF;

     // Edge detection
     #statExecuteOld := #Execute;
   END_REGION

   CASE #statAxisType OF
     #IDLE:
       ;

     #SYNCHRONOUS_AXIS:
         REGION VALID_AXIS
             // Inputs  
             #instMC.Execute := #Execute;

             // Call of MC instruction
             #instMC(Slave := #statAxis);

             // Outputs
             #Done           := #instMC.Done;
             #Busy           := #instMC.Busy;
             #CommandAborted := #instMC.CommandAborted;
             #Error          := #instMC.Error;
             #ErrorID        := #instMC.ErrorId;
             #CoveredOffset  := #instMC.CoveredOffset;
             #StartOffset    := #instMC.StartOffset;

             // Status of MC instruction
             IF NOT #instMC.Done
                 AND NOT #instMC.Busy
                 AND NOT #instMC.CommandAborted
                 AND NOT #instMC.Error
             THEN
                 // Not active
                 #statAxisType := #IDLE;
             END_IF;
         END_REGION

     ELSE
       REGION INVALID_TECHNOLOGY_OBJECT
         // Outputs
         #Done           := FALSE;
         #Busy           := FALSE;
         #CommandAborted := FALSE;
         #Error          := TRUE;
         #ErrorID        := #ERROR_INVALID_TECHNOLOGY_OBJECT;
         #CoveredOffset  := 0.0;
         #StartOffset    := FALSE;
       END_REGION
   END_CASE;
END_FUNCTION_BLOCK

FUNCTION_BLOCK "LAnyAxis_MC_OffsetAbsolute"   // FB30029, SCL
TITLE = LAnyAxis_MC_OffsetAbsolute
{ S7_Optimized_Access := 'TRUE' }
AUTHOR : tech.team.motioncontrol@siemens.com
FAMILY : AnyAxis
VERSION : 1.1
// Support: tech.team.motioncontrol@siemens.com 
// See corresponding MC_ instruction in TIA Portal help (information system)
   VAR_INPUT
      Slave : DB_ANY;   // See corresponding parameter of MC_ instruction in TIA Portal help (information system)
      Execute : Bool;   // See corresponding parameter of MC_ instruction in TIA Portal help (information system)
      Offset : LReal;   // See corresponding parameter of MC_ instruction in TIA Portal help (information system)
      ProfileReference : DInt := 1;   // See corresponding parameter of MC_ instruction in TIA Portal help (information system)
      OffsetDistance : LReal;   // See corresponding parameter of MC_ instruction in TIA Portal help (information system)
      StartPosition : LReal;   // See corresponding parameter of MC_ instruction in TIA Portal help (information system)
      Direction : DInt := 3;   // See corresponding parameter of MC_ instruction in TIA Portal help (information system)
   END_VAR
   VAR_OUTPUT
      Done : Bool;   // See corresponding parameter of MC_ instruction in TIA Portal help (information system)
      Busy : Bool;   // See corresponding parameter of MC_ instruction in TIA Portal help (information system)
      CommandAborted : Bool;   // See corresponding parameter of MC_ instruction in TIA Portal help (information system)
      Error : Bool;   // See corresponding parameter of MC_ instruction in TIA Portal help (information system)
      ErrorID : Word;   // See corresponding parameter of MC_ instruction in TIA Portal help (information system)
      AbsoluteOffset : LReal;   // See corresponding parameter of MC_ instruction in TIA Portal help (information system)
      StartOffset : Bool;   // See corresponding parameter of MC_ instruction in TIA Portal help (information system)
   END_VAR
   VAR
      instMC : MC_OFFSETABSOLUTE;   // Instance of MC_Instruction
      statExecuteOld : Bool;   // Old value of execute
      statAxis : DB_ANY;   // Internal variable of axis
      statAxisType : Int;   // Actual state / axis type
   END_VAR
   VAR CONSTANT
      ERROR_INVALID_TECHNOLOGY_OBJECT : Word := 16#8002;   // See corresponding parameter of MC_ instruction in TIA Portal help (information system)
      IDLE : Int := 0;   // State idle
      INVALID_AXIS : Int := -1;   // Axis type: Invalid
      SYNCHRONOUS_AXIS : Int := 4;   // Axis type: Synchronous axis
   END_VAR
BEGIN
   REGION HEADER
     //================================================================================
     // SIEMENS AG
     // (c)Copyright 2021 All Rights Reserved
     //--------------------------------------------------------------------------------
     // Library: LAnyAxis 
     // Tested with: S7-1515T-2 PN
     // Engineering: TIA Portal V17
     // Restrictions: -
     // Requirements: S7-1500T FW 2.9
     // Functionality: Conversion DB_ANY --> TO_Axis
     // Support: tech.team.motioncontrol@siemens.com
     // Note: Parameter comments are only available in language 'English (United States)'
     //--------------------------------------------------------------------------------
     // Change log table:
     // Version  Date        Expert in charge  Changes applied
     // 01.00.00 01.01.2021  RS                First released version
     // 01.01.00 24.02.2021  RS                Update MC V6.0
     //================================================================================
   END_REGION

   REGION EXECUTE
     IF #Execute AND NOT #statExecuteOld THEN
       // Copy parameter
         #instMC.Offset           := #Offset;
         #instMC.ProfileReference := #ProfileReference;
         #instMC.OffsetDistance   := #OffsetDistance;
         #instMC.StartPosition    := #StartPosition;
         #instMC.Direction        := #Direction;

       // Check axis type
       CASE TypeOfDB(#Slave) OF
         TO_SYNCHRONOUSAXIS:
           #statAxisType := #SYNCHRONOUS_AXIS;
           #statAxis := #Slave;
       ELSE
           #statAxisType := #INVALID_AXIS;
           #statAxis := 0;
       END_CASE;

     ELSIF NOT #Execute AND (#statAxisType < #IDLE) THEN
       #statAxisType := #IDLE;

       // Outputs
       #Done           := FALSE;
       #Busy           := FALSE;
       #CommandAborted := FALSE;
       #Error          := FALSE;
       #ErrorID        := 16#0000;
       #AbsoluteOffset := 0.0;
       #StartOffset    := FALSE;
     END_IF;

     // Edge detection
     #statExecuteOld := #Execute;
   END_REGION

   CASE #statAxisType OF
     #IDLE:
       ;

     #SYNCHRONOUS_AXIS:
         REGION VALID_AXIS
             // Inputs  
             #instMC.Execute := #Execute;

             // Call of MC instruction
             #instMC(Slave := #statAxis);

             // Outputs
             #Done           := #instMC.Done;
             #Busy           := #instMC.Busy;
             #CommandAborted := #instMC.CommandAborted;
             #Error          := #instMC.Error;
             #ErrorID        := #instMC.ErrorId;
             #AbsoluteOffset := #instMC.AbsoluteOffset;
             #StartOffset    := #instMC.StartOffset;

             // Status of MC instruction
             IF NOT #instMC.Done
                 AND NOT #instMC.Busy
                 AND NOT #instMC.CommandAborted
                 AND NOT #instMC.Error
             THEN
                 // Not active
                 #statAxisType := #IDLE;
             END_IF;
         END_REGION

     ELSE
       REGION INVALID_TECHNOLOGY_OBJECT
         // Outputs
         #Done           := FALSE;
         #Busy           := FALSE;
         #CommandAborted := FALSE;
         #Error          := TRUE;
         #ErrorID        := #ERROR_INVALID_TECHNOLOGY_OBJECT;
         #AbsoluteOffset := 0.0;
         #StartOffset    := FALSE;
       END_REGION
   END_CASE;
END_FUNCTION_BLOCK

FUNCTION_BLOCK "LAnyAxis_MC_GearOut"   // FB30032, SCL
TITLE = LAnyAxis_MC_GearOut
{ S7_Optimized_Access := 'TRUE' }
AUTHOR : tech.team.motioncontrol@siemens.com
FAMILY : AnyAxis
VERSION : 1.1
// Support: tech.team.motioncontrol@siemens.com 
// See corresponding MC_ instruction in TIA Portal help (information system)
   VAR_INPUT
      Slave : DB_ANY;   // See corresponding parameter of MC_ instruction in TIA Portal help (information system)
      Execute : Bool;   // See corresponding parameter of MC_ instruction in TIA Portal help (information system)
      SlavePosition : LReal;   // See corresponding parameter of MC_ instruction in TIA Portal help (information system)
      SyncProfileReference : DInt := 1;   // See corresponding parameter of MC_ instruction in TIA Portal help (information system)
      MasterStopDistance : LReal;   // See corresponding parameter of MC_ instruction in TIA Portal help (information system)
      Deceleration : LReal := -1.0;   // See corresponding parameter of MC_ instruction in TIA Portal help (information system)
      Jerk : LReal := -1.0;   // See corresponding parameter of MC_ instruction in TIA Portal help (information system)
      SyncOutDirection : DInt := 3;   // See corresponding parameter of MC_ instruction in TIA Portal help (information system)
   END_VAR
   VAR_OUTPUT
      StartSyncOut : Bool;   // See corresponding parameter of MC_ instruction in TIA Portal help (information system)
      Done : Bool;   // See corresponding parameter of MC_ instruction in TIA Portal help (information system)
      Busy : Bool;   // See corresponding parameter of MC_ instruction in TIA Portal help (information system)
      CommandAborted : Bool;   // See corresponding parameter of MC_ instruction in TIA Portal help (information system)
      Error : Bool;   // See corresponding parameter of MC_ instruction in TIA Portal help (information system)
      ErrorID : Word;   // See corresponding parameter of MC_ instruction in TIA Portal help (information system)
   END_VAR
   VAR
      instMC : MC_GEAROUT;   // Instance of MC_Instruction
      statExecuteOld : Bool;   // Old value of execute
      statAxis : DB_ANY;   // Internal variable of axis
      statAxisType : Int;   // Actual state / axis type
   END_VAR
   VAR CONSTANT
      ERROR_INVALID_TECHNOLOGY_OBJECT : Word := 16#8002;   // See corresponding parameter of MC_ instruction in TIA Portal help (information system)
      IDLE : Int := 0;   // State idle
      INVALID_AXIS : Int := -1;   // Axis type: Invalid
      SYNCHRONOUS_AXIS : Int := 4;   // Axis type: Synchronous axis
   END_VAR
BEGIN
   REGION HEADER
     //================================================================================
     // SIEMENS AG
     // (c)Copyright 2021 All Rights Reserved
     //--------------------------------------------------------------------------------
     // Library: LAnyAxis 
     // Tested with: S7-1515T-2 PN
     // Engineering: TIA Portal V17
     // Restrictions: -
     // Requirements: S7-1500T FW 2.9
     // Functionality: Conversion DB_ANY --> TO_Axis
     // Support: tech.team.motioncontrol@siemens.com
     // Note: Parameter comments are only available in language 'English (United States)'
     //--------------------------------------------------------------------------------
     // Change log table:
     // Version  Date        Expert in charge  Changes applied
     // 01.00.00 10.03.2020  RS                First released version
     // 01.01.00 24.02.2021  RS                Update MC V6.0
     //================================================================================
   END_REGION

   REGION EXECUTE
     IF #Execute AND NOT #statExecuteOld THEN

       // Copy parameter
       #instMC.SlavePosition        := #SlavePosition;
       #instMC.SyncProfileReference := #SyncProfileReference;
       #instMC.MasterStopDistance   := #MasterStopDistance;
       #instMC.Deceleration         := #Deceleration;
       #instMC.Jerk                 := #Jerk;
       #instMC.SyncOutDirection     := #SyncOutDirection;

       // Check axis type
       CASE TypeOfDB(#Slave) OF
         TO_SYNCHRONOUSAXIS:
           #statAxisType := #SYNCHRONOUS_AXIS;
           #statAxis := #Slave;

         ELSE
           #statAxisType := #INVALID_AXIS;
           #statAxis := 0;
       END_CASE;

     ELSIF NOT #Execute AND (#statAxisType < #IDLE) THEN
       #statAxisType := #IDLE;

       // Outputs
       #StartSyncOut   := FALSE;
       #Done           := FALSE;
       #Busy           := FALSE;
       #CommandAborted := FALSE;
       #Error          := FALSE;
       #ErrorID        := 16#0000;
     END_IF;

     // Edge detection
     #statExecuteOld := #Execute;
   END_REGION

   CASE #statAxisType OF
     #IDLE:
       ;

     #SYNCHRONOUS_AXIS:
       REGION VALID_AXIS
         // Inputs
         #instMC.Execute := #Execute;

         // Call of MC instruction
         #instMC(Slave := #statAxis);

         // Outputs
         #StartSyncOut   := #instMC.StartSyncOut;
         #Done           := #instMC.Done;
         #Busy           := #instMC.Busy;
         #CommandAborted := #instMC.CommandAborted;
         #Error          := #instMC.Error;
         #ErrorID        := #instMC.ErrorId;

         // Status of MC instruction
         IF NOT #instMC.Busy
           AND NOT #instMC.CommandAborted
           AND NOT #instMC.Error
           AND NOT #instMC.Done
         THEN
           // Not active
           #statAxisType := #IDLE;
         END_IF;
       END_REGION

     ELSE
       REGION INVALID_TECHNOLOGY_OBJECT
         // Outputs
         #StartSyncOut   := FALSE;
         #Done           := FALSE;
         #Busy           := FALSE;
         #CommandAborted := FALSE;
         #Error          := TRUE;
         #ErrorID        := #ERROR_INVALID_TECHNOLOGY_OBJECT;
       END_REGION
   END_CASE;
END_FUNCTION_BLOCK

FUNCTION_BLOCK "LAnyAxis_MC_CamOut"   // FB30033, SCL
TITLE = LAnyAxis_MC_CamOut
{ S7_Optimized_Access := 'TRUE' }
AUTHOR : tech.team.motioncontrol@siemens.com
FAMILY : AnyAxis
VERSION : 1.1
// Support: tech.team.motioncontrol@siemens.com 
// See corresponding MC_ instruction in TIA Portal help (information system)
   VAR_INPUT
      Slave : DB_ANY;   // See corresponding parameter of MC_ instruction in TIA Portal help (information system)
      Execute : Bool;   // See corresponding parameter of MC_ instruction in TIA Portal help (information system)
      SlavePosition : LReal;   // See corresponding parameter of MC_ instruction in TIA Portal help (information system)
      SyncProfileReference : DInt := 1;   // See corresponding parameter of MC_ instruction in TIA Portal help (information system)
      MasterStopDistance : LReal;   // See corresponding parameter of MC_ instruction in TIA Portal help (information system)
      Deceleration : LReal := -1.0;   // See corresponding parameter of MC_ instruction in TIA Portal help (information system)
      Jerk : LReal := -1.0;   // See corresponding parameter of MC_ instruction in TIA Portal help (information system)
      SyncOutDirection : DInt := 3;   // See corresponding parameter of MC_ instruction in TIA Portal help (information system)
   END_VAR
   VAR_OUTPUT
      StartSyncOut : Bool;   // See corresponding parameter of MC_ instruction in TIA Portal help (information system)
      Done : Bool;   // See corresponding parameter of MC_ instruction in TIA Portal help (information system)
      Busy : Bool;   // See corresponding parameter of MC_ instruction in TIA Portal help (information system)
      CommandAborted : Bool;   // See corresponding parameter of MC_ instruction in TIA Portal help (information system)
      Error : Bool;   // See corresponding parameter of MC_ instruction in TIA Portal help (information system)
      ErrorID : Word;   // See corresponding parameter of MC_ instruction in TIA Portal help (information system)
   END_VAR
   VAR
      instMC : MC_CAMOUT;   // Instance of MC_Instruction
      statExecuteOld : Bool;   // Old value of execute
      statAxis : DB_ANY;   // Internal variable of axis
      statAxisType : Int;   // Actual state / axis type
   END_VAR
   VAR CONSTANT
      ERROR_INVALID_TECHNOLOGY_OBJECT : Word := 16#8002;   // See corresponding parameter of MC_ instruction in TIA Portal help (information system)
      IDLE : Int := 0;   // State idle
      INVALID_AXIS : Int := -1;   // Axis type: Invalid
      SYNCHRONOUS_AXIS : Int := 4;   // Axis type: Synchronous axis
   END_VAR
BEGIN
   REGION HEADER
     //================================================================================
     // SIEMENS AG
     // (c)Copyright 2021 All Rights Reserved
     //--------------------------------------------------------------------------------
     // Library: LAnyAxis 
     // Tested with: S7-1515T-2 PN
     // Engineering: TIA Portal V17
     // Restrictions: -
     // Requirements: S7-1500T FW 2.9
     // Functionality: Conversion DB_ANY --> TO_Axis
     // Support: tech.team.motioncontrol@siemens.com
     // Note: Parameter comments are only available in language 'English (United States)'
     //--------------------------------------------------------------------------------
     // Change log table:
     // Version  Date        Expert in charge  Changes applied
     // 01.00.00 10.03.2020  RS                First released version
     // 01.01.00 24.02.2021  RS                Update MC V6.0
     //================================================================================
   END_REGION

   REGION EXECUTE
     IF #Execute AND NOT #statExecuteOld THEN
       // Copy parameter
       #instMC.SlavePosition        := #SlavePosition;
       #instMC.SyncProfileReference := #SyncProfileReference;
       #instMC.MasterStopDistance   := #MasterStopDistance;
       #instMC.Deceleration         := #Deceleration;
       #instMC.Jerk                 := #Jerk;
       #instMC.SyncOutDirection     := #SyncOutDirection;

       // Check axis type
       CASE TypeOfDB(#Slave) OF
         TO_SYNCHRONOUSAXIS:
           #statAxisType := #SYNCHRONOUS_AXIS;
           #statAxis := #Slave;

         ELSE
           #statAxisType := #INVALID_AXIS;
           #statAxis := 0;
       END_CASE;

     ELSIF NOT #Execute AND (#statAxisType < #IDLE) THEN
       #statAxisType := #IDLE;

       // Outputs
       #StartSyncOut   := FALSE;
       #Done           := FALSE;
       #Busy           := FALSE;
       #CommandAborted := FALSE;
       #Error          := FALSE;
       #ErrorID        := 16#0000;
     END_IF;

     // Edge detection
     #statExecuteOld := #Execute;
   END_REGION

   CASE #statAxisType OF
     #IDLE:
       ;

     #SYNCHRONOUS_AXIS:
       REGION VALID_AXIS
         // Inputs
         #instMC.Execute := #Execute;

         // Call of MC instruction
         #instMC(Slave := #statAxis);

         // Outputs
         #StartSyncOut   := #instMC.StartSyncOut;
         #Done           := #instMC.Done;
         #Busy           := #instMC.Busy;
         #CommandAborted := #instMC.CommandAborted;
         #Error          := #instMC.Error;
         #ErrorID        := #instMC.ErrorId;

         // Status of MC instruction
         IF NOT #instMC.Busy
           AND NOT #instMC.CommandAborted
           AND NOT #instMC.Error
           AND NOT #instMC.Done
         THEN
           // Not active
           #statAxisType := #IDLE;
         END_IF;
       END_REGION

     ELSE
       REGION INVALID_TECHNOLOGY_OBJECT
         // Outputs
         #StartSyncOut   := FALSE;
         #Done           := FALSE;
         #Busy           := FALSE;
         #CommandAborted := FALSE;
         #Error          := TRUE;
         #ErrorID        := #ERROR_INVALID_TECHNOLOGY_OBJECT;
       END_REGION
   END_CASE;
END_FUNCTION_BLOCK

// folder: LAnyAxis_Blocks/LAnyAxis_MC_SynchronousMotion/InternalSubBlocks/MC_CamIn

FUNCTION "LAnyAxis_UnpubCamInMasterExtEncoder" : Void   // FC30037, SCL
TITLE = LAnyAxis_UnpubCamInMasterExtEncoder
{ S7_Optimized_Access := 'TRUE' }
AUTHOR : tech.team.motioncontrol@siemens.com
FAMILY : AnyAxis
VERSION : 1.0
// Support: tech.team.motioncontrol@siemens.com
   VAR_INPUT
      slave : TO_SynchronousAxis;   // Slave axis specification
      master : TO_ExternalEncoder;   // Master axis specification
      cam : TO_Cam;   // Cam specification
   END_VAR
   VAR_IN_OUT
      instMC : MC_CAMIN;   // Instance of MC_Instruction
   END_VAR
   // Ret_Val : No return value
BEGIN
   // Call of MC_Instruction
   #instMC(Master := #master,
           Slave := #slave,
           Cam := #cam);
END_FUNCTION

FUNCTION "LAnyAxis_UnpubCamInMasterPosAxis" : Void   // FC30038, SCL
TITLE = LAnyAxis_UnpubCamInMasterPosAxis
{ S7_Optimized_Access := 'TRUE' }
AUTHOR : tech.team.motioncontrol@siemens.com
FAMILY : AnyAxis
VERSION : 1.0
// Support: tech.team.motioncontrol@siemens.com
   VAR_INPUT
      slave : TO_SynchronousAxis;   // Slave axis specification
      master : TO_PositioningAxis;   // Master axis specification
      cam : TO_Cam;   // Cam specification
   END_VAR
   VAR_IN_OUT
      instMC : MC_CAMIN;   // Instance of MC_Instruction
   END_VAR
   // Ret_Val : No return value
BEGIN
   // Call of MC_Instruction
   #instMC(Master := #master,
           Slave := #slave,
           Cam := #cam);
END_FUNCTION

FUNCTION "LAnyAxis_UnpubCamInMasterProxy" : Void   // FC30039, SCL
TITLE = LAnyAxis_UnpubCamInMasterProxy
{ S7_Optimized_Access := 'TRUE' }
AUTHOR : tech.team.motioncontrol@siemens.com
FAMILY : AnyAxis
VERSION : 1.0
// Support: tech.team.motioncontrol@siemens.com
   VAR_INPUT
      slave : TO_SynchronousAxis;   // Slave axis specification
      master : TO_LeadingAxisProxy;   // Master axis specification
      cam : TO_Cam;   // Cam specification
   END_VAR
   VAR_IN_OUT
      instMC : MC_CAMIN;   // Instance of MC_Instruction
   END_VAR
   // Ret_Val : No return value
BEGIN
   // Call of MC_Instruction
   #instMC(Master := #master,
           Slave := #slave,
           Cam := #cam);
END_FUNCTION

FUNCTION "LAnyAxis_UnpubCamInMasterSyncAxis" : Void   // FC30040, SCL
TITLE = LAnyAxis_UnpubCamInMasterSyncAxis
{ S7_Optimized_Access := 'TRUE' }
AUTHOR : tech.team.motioncontrol@siemens.com
FAMILY : AnyAxis
VERSION : 1.0
// Support: tech.team.motioncontrol@siemens.com
   VAR_INPUT
      slave : TO_SynchronousAxis;   // Slave axis specification
      master : TO_SynchronousAxis;   // Master axis specification
      cam : TO_Cam;   // Cam specification
   END_VAR
   VAR_IN_OUT
      instMC : MC_CAMIN;   // Instance of MC_Instruction
   END_VAR
   // Ret_Val : No return value
BEGIN
   // Call of MC_Instruction
   #instMC(Master := #master,
           Slave := #slave,
           Cam := #cam);
END_FUNCTION

FUNCTION "LAnyAxis_UnpubCamIn10kMasterExtEncoder" : Void   // FC30056, SCL
TITLE = LAnyAxis_UnpubCamIn10kMasterExtEncoder
{ S7_Optimized_Access := 'TRUE' }
AUTHOR : tech.team.motioncontrol@siemens.com
FAMILY : AnyAxis
VERSION : 1.0
// Support: tech.team.motioncontrol@siemens.com
   VAR_INPUT
      slave : TO_SynchronousAxis;   // Slave axis specification
      master : TO_ExternalEncoder;   // Master axis specification
      cam : TO_Cam_10k;   // Cam specification
   END_VAR
   VAR_IN_OUT
      instMC : MC_CAMIN;   // Instance of MC_Instruction
   END_VAR
   // Ret_Val : No return value
BEGIN
   // Call of MC_Instruction
   #instMC(Master := #master,
           Slave := #slave,
           Cam := #cam);
END_FUNCTION

FUNCTION "LAnyAxis_UnpubCamIn10kMasterPosAxis" : Void   // FC30082, SCL
TITLE = LAnyAxis_UnpubCamIn10kMasterPosAxis
{ S7_Optimized_Access := 'TRUE' }
AUTHOR : tech.team.motioncontrol@siemens.com
FAMILY : AnyAxis
VERSION : 1.0
// Support: tech.team.motioncontrol@siemens.com
   VAR_INPUT
      slave : TO_SynchronousAxis;   // Slave axis specification
      master : TO_PositioningAxis;   // Master axis specification
      cam : TO_Cam_10k;   // Cam specification
   END_VAR
   VAR_IN_OUT
      instMC : MC_CAMIN;   // Instance of MC_Instruction
   END_VAR
   // Ret_Val : No return value
BEGIN
   // Call of MC_Instruction
   #instMC(Master := #master,
           Slave  := #slave,
           Cam    := #cam);
END_FUNCTION

FUNCTION "LAnyAxis_UnpubCamIn10kMasterProxy" : Void   // FC30083, SCL
TITLE = LAnyAxis_UnpubCamIn10kMasterProxy
{ S7_Optimized_Access := 'TRUE' }
AUTHOR : tech.team.motioncontrol@siemens.com
FAMILY : AnyAxis
VERSION : 1.0
// Support: tech.team.motioncontrol@siemens.com
   VAR_INPUT
      slave : TO_SynchronousAxis;   // Slave axis specification
      master : TO_LeadingAxisProxy;   // Master axis specification
      cam : TO_Cam_10k;   // Cam specification
   END_VAR
   VAR_IN_OUT
      instMC : MC_CAMIN;   // Instance of MC_Instruction
   END_VAR
   // Ret_Val : No return value
BEGIN
   // Call of MC_Instruction
   #instMC(Master := #master,
           Slave := #slave,
           Cam := #cam);
END_FUNCTION

FUNCTION "LAnyAxis_UnpubCamIn10kMasterSyncAxis" : Void   // FC30084, SCL
TITLE = LAnyAxis_UnpubCamIn10kMasterSyncAxis
{ S7_Optimized_Access := 'TRUE' }
AUTHOR : tech.team.motioncontrol@siemens.com
FAMILY : AnyAxis
VERSION : 1.0
// Support: tech.team.motioncontrol@siemens.com
   VAR_INPUT
      slave : TO_SynchronousAxis;   // Slave axis specification
      master : TO_SynchronousAxis;   // Master axis specification
      cam : TO_Cam_10k;   // Cam specification
   END_VAR
   VAR_IN_OUT
      instMC : MC_CAMIN;   // Instance of MC_Instruction
   END_VAR
   // Ret_Val : No return value
BEGIN
   // Call of MC_Instruction
   #instMC(Master := #master,
           Slave := #slave,
           Cam := #cam);
END_FUNCTION

// folder: LAnyAxis_Blocks/LAnyAxis_MC_SynchronousMotion/InternalSubBlocks/MC_GearIn

FUNCTION "LAnyAxis_UnpubGearInMasterExtEncoder" : Void   // FC30000, SCL
TITLE = LAnyAxis_UnpubGearInMasterExtEncoder
{ S7_Optimized_Access := 'TRUE' }
AUTHOR : tech.team.motioncontrol@siemens.com
FAMILY : AnyAxis
VERSION : 1.0
// Support: tech.team.motioncontrol@siemens.com
   VAR_INPUT
      slave : TO_SynchronousAxis;   // Slave axis specification
      master : TO_ExternalEncoder;   // Master axis specification
   END_VAR
   VAR_IN_OUT
      instMC : MC_GEARIN;   // Instance of MC_Instruction
   END_VAR
   // Ret_Val : No return value
BEGIN
   // Call of MC_Instruction
   #instMC(Master := #master,
           Slave := #slave);
END_FUNCTION

FUNCTION "LAnyAxis_UnpubGearInMasterPosAxis" : Void   // FC30001, SCL
TITLE = LAnyAxis_UnpubGearInMasterPosAxis
{ S7_Optimized_Access := 'TRUE' }
AUTHOR : tech.team.motioncontrol@siemens.com
FAMILY : AnyAxis
VERSION : 1.0
// Support: tech.team.motioncontrol@siemens.com
   VAR_INPUT
      slave : TO_SynchronousAxis;   // Slave axis specification
      master : TO_PositioningAxis;   // Master axis specification
   END_VAR
   VAR_IN_OUT
      instMC : MC_GEARIN;   // Instance of MC_Instruction
   END_VAR
   // Ret_Val : No return value
BEGIN
   // Call of MC_Instruction
   #instMC(Master := #master,
           Slave := #slave);
END_FUNCTION

FUNCTION "LAnyAxis_UnpubGearInMasterSyncAxis" : Void   // FC30002, SCL
TITLE = LAnyAxis_UnpubGearInMasterSyncAxis
{ S7_Optimized_Access := 'TRUE' }
AUTHOR : tech.team.motioncontrol@siemens.com
FAMILY : AnyAxis
VERSION : 1.0
// Support: tech.team.motioncontrol@siemens.com
   VAR_INPUT
      slave : TO_SynchronousAxis;   // Slave axis specification
      master : TO_SynchronousAxis;   // Master axis specification
   END_VAR
   VAR_IN_OUT
      instMC : MC_GEARIN;   // Instance of MC_Instruction
   END_VAR
   // Ret_Val : No return value
BEGIN
   // Call of MC_Instruction
   #instMC(Master := #master,
           Slave := #slave);
END_FUNCTION

FUNCTION "LAnyAxis_UnpubGearInMasterProxy" : Void   // FC30041, SCL
TITLE = LAnyAxis_UnpubGearInMasterProxy
{ S7_Optimized_Access := 'TRUE' }
AUTHOR : tech.team.motioncontrol@siemens.com
FAMILY : AnyAxis
VERSION : 1.0
// Support: tech.team.motioncontrol@siemens.com
   VAR_INPUT
      slave : TO_SynchronousAxis;   // Slave axis specification
      master : TO_LeadingAxisProxy;   // Master axis specification
   END_VAR
   VAR_IN_OUT
      instMC : MC_GEARIN;   // Instance of MC_Instruction
   END_VAR
   // Ret_Val : No return value
BEGIN
   // Call of MC_Instruction
   #instMC(Master := #master,
           Slave := #slave);
END_FUNCTION

// folder: LAnyAxis_Blocks/LAnyAxis_MC_SynchronousMotion/InternalSubBlocks/MC_GearInPos

FUNCTION "LAnyAxis_UnpubGearInPosMasterExtEncoder" : Void   // FC30044, SCL
TITLE = LAnyAxis_UnpubGearInPosMasterExtEncoder
{ S7_Optimized_Access := 'TRUE' }
AUTHOR : tech.team.motioncontrol@siemens.com
FAMILY : AnyAxis
VERSION : 1.0
// Support: tech.team.motioncontrol@siemens.com
   VAR_INPUT
      slave : TO_SynchronousAxis;   // Slave axis specification
      master : TO_ExternalEncoder;   // Master axis specification
   END_VAR
   VAR_IN_OUT
      instMC : MC_GEARINPOS;   // Instance of MC_Instruction
   END_VAR
   // Ret_Val : No return value
BEGIN
   // Call of MC_Instruction
   #instMC(Master := #master,
           Slave := #slave);
END_FUNCTION

FUNCTION "LAnyAxis_UnpubGearInPosMasterPosAxis" : Void   // FC30045, SCL
TITLE = LAnyAxis_UnpubGearInPosMasterPosAxis
{ S7_Optimized_Access := 'TRUE' }
AUTHOR : tech.team.motioncontrol@siemens.com
FAMILY : AnyAxis
VERSION : 1.0
// Support: tech.team.motioncontrol@siemens.com
   VAR_INPUT
      slave : TO_SynchronousAxis;   // Slave axis specification
      master : TO_PositioningAxis;   // Master axis specification
   END_VAR
   VAR_IN_OUT
      instMC : MC_GEARINPOS;   // Instance of MC_Instruction
   END_VAR
   // Ret_Val : No return value
BEGIN
   // Call of MC_Instruction
   #instMC(Master := #master,
           Slave := #slave);
END_FUNCTION

FUNCTION "LAnyAxis_UnpubGearInPosMasterProxy" : Void   // FC30046, SCL
TITLE = LAnyAxis_UnpubGearInPosMasterProxy
{ S7_Optimized_Access := 'TRUE' }
AUTHOR : tech.team.motioncontrol@siemens.com
FAMILY : AnyAxis
VERSION : 1.0
// Support: tech.team.motioncontrol@siemens.com
   VAR_INPUT
      slave : TO_SynchronousAxis;   // Slave axis specification
      master : TO_LeadingAxisProxy;   // Master axis specification
   END_VAR
   VAR_IN_OUT
      instMC : MC_GEARINPOS;   // Instance of MC_Instruction
   END_VAR
   // Ret_Val : No return value
BEGIN
   // Call of MC_Instruction
   #instMC(Master := #master,
           Slave := #slave);
END_FUNCTION

FUNCTION "LAnyAxis_UnpubGearInPosMasterSyncAxis" : Void   // FC30047, SCL
TITLE = LAnyAxis_UnpubGearInPosMasterSyncAxis
{ S7_Optimized_Access := 'TRUE' }
AUTHOR : tech.team.motioncontrol@siemens.com
FAMILY : AnyAxis
VERSION : 1.0
// Support: tech.team.motioncontrol@siemens.com
   VAR_INPUT
      slave : TO_SynchronousAxis;   // Slave axis specification
      master : TO_SynchronousAxis;   // Master axis specification
   END_VAR
   VAR_IN_OUT
      instMC : MC_GEARINPOS;   // Instance of MC_Instruction
   END_VAR
   // Ret_Val : No return value
BEGIN
   // Call of MC_Instruction
   #instMC(Master := #master,
           Slave := #slave);
END_FUNCTION

// folder: LAnyAxis_Blocks/LAnyAxis_MC_SynchronousMotion/InternalSubBlocks/MC_PhasingAbsolute

FUNCTION "LAnyAxis_UnpubPhasingAbsoluteMasterExtEncoder" : Void   // FC30048, SCL
TITLE = LAnyAxis_UnpubPhasingAbsoluteMasterExtEncoder
{ S7_Optimized_Access := 'TRUE' }
AUTHOR : tech.team.motioncontrol@siemens.com
FAMILY : AnyAxis
VERSION : 1.0
// Support: tech.team.motioncontrol@siemens.com
   VAR_INPUT
      slave : TO_SynchronousAxis;   // Slave axis specification
      master : TO_ExternalEncoder;   // Master axis specification
   END_VAR
   VAR_IN_OUT
      instMC : MC_PHASINGABSOLUTE;   // Instance of MC_Instruction
   END_VAR
   // Ret_Val : No return value
BEGIN
   // Call of MC_Instruction
   #instMC(Master := #master,
           Slave := #slave);
END_FUNCTION

FUNCTION "LAnyAxis_UnpubPhasingAbsoluteMasterPosAxis" : Void   // FC30049, SCL
TITLE = LAnyAxis_UnpubPhasingAbsoluteMasterPosAxis
{ S7_Optimized_Access := 'TRUE' }
AUTHOR : tech.team.motioncontrol@siemens.com
FAMILY : AnyAxis
VERSION : 1.0
// Support: tech.team.motioncontrol@siemens.com
   VAR_INPUT
      slave : TO_SynchronousAxis;   // Slave axis specification
      master : TO_PositioningAxis;   // Master axis specification
   END_VAR
   VAR_IN_OUT
      instMC : MC_PHASINGABSOLUTE;   // Instance of MC_Instruction
   END_VAR
   // Ret_Val : No return value
BEGIN
   // Call of MC_Instruction
   #instMC(Master := #master,
           Slave := #slave);
END_FUNCTION

FUNCTION "LAnyAxis_UnpubPhasingAbsoluteMasterProxy" : Void   // FC30050, SCL
TITLE = LAnyAxis_UnpubPhasingAbsoluteMasterProxy
{ S7_Optimized_Access := 'TRUE' }
AUTHOR : tech.team.motioncontrol@siemens.com
FAMILY : AnyAxis
VERSION : 1.0
// Support: tech.team.motioncontrol@siemens.com
   VAR_INPUT
      slave : TO_SynchronousAxis;   // Slave axis specification
      master : TO_LeadingAxisProxy;   // Master axis specification
   END_VAR
   VAR_IN_OUT
      instMC : MC_PHASINGABSOLUTE;   // Instance of MC_Instruction
   END_VAR
   // Ret_Val : No return value
BEGIN
   // Call of MC_Instruction
   #instMC(Master := #master,
           Slave := #slave);
END_FUNCTION

FUNCTION "LAnyAxis_UnpubPhasingAbsoluteMasterSyncAxis" : Void   // FC30051, SCL
TITLE = LAnyAxis_UnpubPhasingAbsoluteMasterSyncAxis
{ S7_Optimized_Access := 'TRUE' }
AUTHOR : tech.team.motioncontrol@siemens.com
FAMILY : AnyAxis
VERSION : 1.0
// Support: tech.team.motioncontrol@siemens.com
   VAR_INPUT
      slave : TO_SynchronousAxis;   // Slave axis specification
      master : TO_SynchronousAxis;   // Master axis specification
   END_VAR
   VAR_IN_OUT
      instMC : MC_PHASINGABSOLUTE;   // Instance of MC_Instruction
   END_VAR
   // Ret_Val : No return value
BEGIN
   // Call of MC_Instruction
   #instMC(Master := #master,
           Slave := #slave);
END_FUNCTION

// folder: LAnyAxis_Blocks/LAnyAxis_MC_SynchronousMotion/InternalSubBlocks/MC_PhasingRelative

FUNCTION "LAnyAxis_UnpubPhasingRelativeMasterExtEncoder" : Void   // FC30052, SCL
TITLE = LAnyAxis_UnpubPhasingRelativeMasterExtEncoder
{ S7_Optimized_Access := 'TRUE' }
AUTHOR : tech.team.motioncontrol@siemens.com
FAMILY : AnyAxis
VERSION : 1.0
// Support: tech.team.motioncontrol@siemens.com
   VAR_INPUT
      slave : TO_SynchronousAxis;   // Slave axis specification
      master : TO_ExternalEncoder;   // Master axis specification
   END_VAR
   VAR_IN_OUT
      instMC : MC_PHASINGRELATIVE;   // Instance of MC_Instruction
   END_VAR
   // Ret_Val : No return value
BEGIN
   // Call of MC_Instruction
   #instMC(Master := #master,
           Slave := #slave);
END_FUNCTION

FUNCTION "LAnyAxis_UnpubPhasingRelativeMasterPosAxis" : Void   // FC30053, SCL
TITLE = LAnyAxis_UnpubPhasingRelativeMasterPosAxis
{ S7_Optimized_Access := 'TRUE' }
AUTHOR : tech.team.motioncontrol@siemens.com
FAMILY : AnyAxis
VERSION : 1.0
// Support: tech.team.motioncontrol@siemens.com
   VAR_INPUT
      slave : TO_SynchronousAxis;   // Slave axis specification
      master : TO_PositioningAxis;   // Master axis specification
   END_VAR
   VAR_IN_OUT
      instMC : MC_PHASINGRELATIVE;   // Instance of MC_Instruction
   END_VAR
   // Ret_Val : No return value
BEGIN
   // Call of MC_Instruction
   #instMC(Master := #master,
           Slave := #slave);
END_FUNCTION

